LIN {X 14.324,Y -289.646,Z 149.698,A 92.831,B 90.000,C 0.000} C_DIS
LIN {X 14.364,Y -289.644,Z 149.777,A 92.839,B 90.000,C 0.000} C_DIS
LIN {X 14.595,Y -289.632,Z 150.119,A 92.885,B 90.000,C 0.000} C_DIS
LIN {X 14.694,Y -289.627,Z 150.212,A 92.904,B 90.000,C 0.000} C_DIS
LIN {X 14.908,Y -289.617,Z 150.520,A 92.947,B 90.000,C 0.000} C_DIS
LIN {X 16.420,Y -289.535,Z 152.509,A 93.246,B 90.000,C 0.000} C_DIS
LIN {X 16.512,Y -289.530,Z 152.653,A 93.264,B 90.000,C 0.000} C_DIS
LIN {X 18.087,Y -289.435,Z 154.593,A 93.576,B 90.000,C 0.000} C_DIS
LIN {X 18.457,Y -289.412,Z 155.070,A 93.649,B 90.000,C 0.000} C_DIS
LIN {X 18.491,Y -289.410,Z 155.103,A 93.656,B 90.000,C 0.000} C_DIS
LIN {X 18.557,Y -289.406,Z 155.188,A 93.669,B 90.000,C 0.000} C_DIS
LIN {X 18.610,Y -289.402,Z 155.273,A 93.679,B 90.000,C 0.000} C_DIS
LIN {X 18.698,Y -289.397,Z 155.384,A 93.697,B 90.000,C 0.000} C_DIS
LIN {X 18.848,Y -289.387,Z 155.532,A 93.726,B 90.000,C 0.000} C_DIS
LIN {X 18.933,Y -289.381,Z 155.598,A 93.743,B 90.000,C 0.000} C_DIS
LIN {X 18.971,Y -289.379,Z 155.701,A 93.751,B 90.000,C 0.000} C_DIS
LIN {X 20.031,Y -289.307,Z 156.976,A 93.961,B 90.000,C 0.000} C_DIS
LIN {X 20.180,Y -289.297,Z 157.094,A 93.990,B 90.000,C 0.000} C_DIS
LIN {X 20.232,Y -289.293,Z 157.151,A 94.000,B 90.000,C 0.000} C_DIS
LIN {X 20.247,Y -289.292,Z 157.208,A 94.004,B 90.000,C 0.000} C_DIS
LIN {X 20.626,Y -289.266,Z 157.610,A 94.079,B 90.000,C 0.000} C_DIS
LIN {X 20.742,Y -289.257,Z 157.720,A 94.102,B 90.000,C 0.000} C_DIS
LIN {X 20.768,Y -289.255,Z 157.777,A 94.107,B 90.000,C 0.000} C_DIS
LIN {X 21.906,Y -289.171,Z 158.799,A 94.332,B 90.000,C 0.000} C_DIS
LIN {X 22.359,Y -289.137,Z 159.201,A 94.422,B 90.000,C 0.000} C_DIS
LIN {X 23.494,Y -289.047,Z 160.165,A 94.647,B 90.000,C 0.000} C_DIS
LIN {X 23.807,Y -289.021,Z 160.394,A 94.709,B 90.000,C 0.000} C_DIS
LIN {X 23.862,Y -289.017,Z 160.451,A 94.720,B 90.000,C 0.000} C_DIS
LIN {X 23.876,Y -289.015,Z 160.508,A 94.723,B 90.000,C 0.000} C_DIS
LIN {X 24.686,Y -288.947,Z 161.134,A 94.883,B 90.000,C 0.000} C_DIS
LIN {X 24.833,Y -288.935,Z 161.286,A 94.912,B 90.000,C 0.000} C_DIS
LIN {X 25.476,Y -288.879,Z 161.759,A 95.040,B 90.000,C 0.000} C_DIS
LIN {X 25.535,Y -288.874,Z 161.845,A 95.051,B 90.000,C 0.000} C_DIS
LIN {X 25.733,Y -288.856,Z 161.987,A 95.091,B 90.000,C 0.000} C_DIS
LIN {X 25.749,Y -288.855,Z 162.044,A 95.094,B 90.000,C 0.000} C_DIS
LIN {X 26.204,Y -288.814,Z 162.384,A 95.184,B 90.000,C 0.000} C_DIS
LIN {X 26.243,Y -288.810,Z 162.442,A 95.192,B 90.000,C 0.000} C_DIS
LIN {X 26.264,Y -288.808,Z 162.499,A 95.196,B 90.000,C 0.000} C_DIS
LIN {X 27.201,Y -288.721,Z 163.333,A 95.382,B 90.000,C 0.000} C_DIS
LIN {X 29.132,Y -288.533,Z 164.205,A 95.765,B 90.000,C 0.000} C_DIS
LIN {X 31.516,Y -288.282,Z 164.913,A 96.239,B 90.000,C 0.000} C_DIS
LIN {X 33.522,Y -288.056,Z 165.228,A 96.638,B 90.000,C 0.000} C_DIS
LIN {X 36.003,Y -287.754,Z 165.278,A 97.132,B 90.000,C 0.000} C_DIS
LIN {X 37.185,Y -287.606,Z 165.298,A 97.367,B 90.000,C 0.000} C_DIS
LIN {X 38.173,Y -287.477,Z 165.175,A 97.564,B 90.000,C 0.000} C_DIS
LIN {X 39.512,Y -287.296,Z 164.884,A 97.831,B 90.000,C 0.000} C_DIS
LIN {X 39.611,Y -287.282,Z 164.845,A 97.850,B 90.000,C 0.000} C_DIS
LIN {X 40.343,Y -287.180,Z 164.702,A 97.997,B 90.000,C 0.000} C_DIS
LIN {X 40.569,Y -287.148,Z 164.621,A 98.042,B 90.000,C 0.000} C_DIS
LIN {X 40.681,Y -287.132,Z 164.611,A 98.064,B 90.000,C 0.000} C_DIS
LIN {X 42.877,Y -286.813,Z 163.977,A 98.502,B 90.000,C 0.000} C_DIS
LIN {X 42.990,Y -286.796,Z 163.962,A 98.525,B 90.000,C 0.000} C_DIS
LIN {X 43.102,Y -286.779,Z 163.932,A 98.547,B 90.000,C 0.000} C_DIS
LIN {X 43.758,Y -286.680,Z 163.656,A 98.678,B 90.000,C 0.000} C_DIS
LIN {X 43.856,Y -286.665,Z 163.644,A 98.698,B 90.000,C 0.000} C_DIS
LIN {X 46.143,Y -286.306,Z 162.699,A 99.155,B 90.000,C 0.000} C_DIS
LIN {X 46.563,Y -286.237,Z 162.499,A 99.240,B 90.000,C 0.000} C_DIS
LIN {X 47.119,Y -286.147,Z 162.115,A 99.351,B 90.000,C 0.000} C_DIS
LIN {X 47.257,Y -286.124,Z 162.044,A 99.378,B 90.000,C 0.000} C_DIS
LIN {X 47.317,Y -286.114,Z 161.984,A 99.391,B 90.000,C 0.000} C_DIS
LIN {X 48.334,Y -285.944,Z 161.191,A 99.594,B 90.000,C 0.000} C_DIS
LIN {X 48.383,Y -285.935,Z 161.105,A 99.604,B 90.000,C 0.000} C_DIS
LIN {X 48.468,Y -285.921,Z 161.020,A 99.621,B 90.000,C 0.000} C_DIS
LIN {X 48.552,Y -285.907,Z 160.953,A 99.638,B 90.000,C 0.000} C_DIS
LIN {X 48.585,Y -285.901,Z 160.921,A 99.644,B 90.000,C 0.000} C_DIS
LIN {X 50.411,Y -285.585,Z 159.243,A 100.011,B 90.000,C 0.000} C_DIS
LIN {X 50.514,Y -285.567,Z 159.135,A 100.031,B 90.000,C 0.000} C_DIS
LIN {X 50.570,Y -285.557,Z 159.114,A 100.043,B 90.000,C 0.000} C_DIS
LIN {X 50.626,Y -285.547,Z 159.064,A 100.054,B 90.000,C 0.000} C_DIS
LIN {X 51.727,Y -285.349,Z 156.829,A 100.275,B 90.000,C 0.000} C_DIS
LIN {X 51.777,Y -285.340,Z 156.731,A 100.285,B 90.000,C 0.000} C_DIS
LIN {X 52.198,Y -285.264,Z 155.800,A 100.369,B 90.000,C 0.000} C_DIS
LIN {X 52.229,Y -285.258,Z 155.405,A 100.376,B 90.000,C 0.000} C_DIS
LIN {X 52.149,Y -285.273,Z 155.422,A 100.359,B 90.000,C 0.000} C_DIS
LIN {X 51.928,Y -285.313,Z 155.589,A 100.315,B 90.000,C 0.000} C_DIS
LIN {X 51.746,Y -285.346,Z 155.763,A 100.279,B 90.000,C 0.000} C_DIS
LIN {X 51.520,Y -285.387,Z 156.070,A 100.233,B 90.000,C 0.000} C_DIS
LIN {X 51.426,Y -285.404,Z 156.169,A 100.214,B 90.000,C 0.000} C_DIS
LIN {X 51.130,Y -285.457,Z 156.551,A 100.155,B 90.000,C 0.000} C_DIS
LIN {X 50.883,Y -285.501,Z 156.767,A 100.105,B 90.000,C 0.000} C_DIS
LIN {X 50.632,Y -285.546,Z 157.151,A 100.055,B 90.000,C 0.000} C_DIS
LIN {X 48.944,Y -285.840,Z 158.739,A 99.717,B 90.000,C 0.000} C_DIS
LIN {X 48.327,Y -285.945,Z 159.090,A 99.593,B 90.000,C 0.000} C_DIS
LIN {X 48.215,Y -285.964,Z 159.139,A 99.570,B 90.000,C 0.000} C_DIS
LIN {X 48.131,Y -285.978,Z 159.199,A 99.554,B 90.000,C 0.000} C_DIS
LIN {X 48.047,Y -285.992,Z 159.243,A 99.537,B 90.000,C 0.000} C_DIS
LIN {X 47.103,Y -286.149,Z 159.921,A 99.348,B 90.000,C 0.000} C_DIS
LIN {X 46.868,Y -286.188,Z 160.040,A 99.301,B 90.000,C 0.000} C_DIS
LIN {X 46.475,Y -286.252,Z 160.349,A 99.222,B 90.000,C 0.000} C_DIS
LIN {X 46.419,Y -286.261,Z 160.366,A 99.211,B 90.000,C 0.000} C_DIS
LIN {X 46.363,Y -286.270,Z 160.391,A 99.199,B 90.000,C 0.000} C_DIS
LIN {X 46.283,Y -286.283,Z 160.451,A 99.183,B 90.000,C 0.000} C_DIS
LIN {X 45.576,Y -286.396,Z 160.853,A 99.042,B 90.000,C 0.000} C_DIS
LIN {X 44.677,Y -286.538,Z 161.257,A 98.862,B 90.000,C 0.000} C_DIS
LIN {X 44.565,Y -286.555,Z 161.295,A 98.840,B 90.000,C 0.000} C_DIS
LIN {X 43.565,Y -286.709,Z 161.759,A 98.640,B 90.000,C 0.000} C_DIS
LIN {X 41.526,Y -287.011,Z 162.566,A 98.233,B 90.000,C 0.000} C_DIS
LIN {X 41.301,Y -287.044,Z 162.601,A 98.188,B 90.000,C 0.000} C_DIS
LIN {X 40.977,Y -287.090,Z 162.722,A 98.123,B 90.000,C 0.000} C_DIS
LIN {X 38.530,Y -287.429,Z 163.103,A 97.635,B 90.000,C 0.000} C_DIS
LIN {X 37.750,Y -287.533,Z 163.175,A 97.480,B 90.000,C 0.000} C_DIS
LIN {X 35.270,Y -287.846,Z 163.117,A 96.986,B 90.000,C 0.000} C_DIS
LIN {X 32.811,Y -288.137,Z 162.780,A 96.496,B 90.000,C 0.000} C_DIS
LIN {X 30.430,Y -288.399,Z 162.061,A 96.023,B 90.000,C 0.000} C_DIS
LIN {X 29.103,Y -288.536,Z 161.533,A 95.760,B 90.000,C 0.000} C_DIS
LIN {X 28.948,Y -288.552,Z 161.424,A 95.729,B 90.000,C 0.000} C_DIS
LIN {X 28.296,Y -288.616,Z 161.071,A 95.599,B 90.000,C 0.000} C_DIS
LIN {X 28.141,Y -288.631,Z 160.962,A 95.569,B 90.000,C 0.000} C_DIS
LIN {X 27.574,Y -288.686,Z 160.678,A 95.456,B 90.000,C 0.000} C_DIS
LIN {X 27.006,Y -288.740,Z 160.337,A 95.343,B 90.000,C 0.000} C_DIS
LIN {X 26.825,Y -288.757,Z 160.259,A 95.307,B 90.000,C 0.000} C_DIS
LIN {X 26.623,Y -288.775,Z 160.142,A 95.267,B 90.000,C 0.000} C_DIS
LIN {X 26.439,Y -288.792,Z 159.996,A 95.231,B 90.000,C 0.000} C_DIS
LIN {X 25.672,Y -288.861,Z 159.484,A 95.079,B 90.000,C 0.000} C_DIS
LIN {X 25.308,Y -288.894,Z 159.140,A 95.007,B 90.000,C 0.000} C_DIS
LIN {X 24.741,Y -288.943,Z 158.391,A 94.894,B 90.000,C 0.000} C_DIS
LIN {X 24.666,Y -288.949,Z 158.346,A 94.879,B 90.000,C 0.000} C_DIS
LIN {X 23.494,Y -289.047,Z 157.203,A 94.647,B 90.000,C 0.000} C_DIS
LIN {X 22.038,Y -289.161,Z 155.956,A 94.358,B 90.000,C 0.000} C_DIS
LIN {X 21.452,Y -289.206,Z 155.331,A 94.242,B 90.000,C 0.000} C_DIS
LIN {X 21.337,Y -289.214,Z 155.245,A 94.219,B 90.000,C 0.000} C_DIS
LIN {X 21.256,Y -289.220,Z 155.155,A 94.203,B 90.000,C 0.000} C_DIS
LIN {X 21.228,Y -289.222,Z 155.103,A 94.198,B 90.000,C 0.000} C_DIS
LIN {X 21.168,Y -289.226,Z 155.043,A 94.186,B 90.000,C 0.000} C_DIS
LIN {X 20.955,Y -289.242,Z 154.735,A 94.144,B 90.000,C 0.000} C_DIS
LIN {X 20.884,Y -289.247,Z 154.595,A 94.130,B 90.000,C 0.000} C_DIS
LIN {X 20.824,Y -289.251,Z 154.534,A 94.118,B 90.000,C 0.000} C_DIS
LIN {X 20.799,Y -289.253,Z 154.477,A 94.113,B 90.000,C 0.000} C_DIS
LIN {X 20.786,Y -289.254,Z 154.420,A 94.110,B 90.000,C 0.000} C_DIS
LIN {X 20.630,Y -289.265,Z 154.235,A 94.079,B 90.000,C 0.000} C_DIS
LIN {X 19.990,Y -289.310,Z 153.410,A 93.953,B 90.000,C 0.000} C_DIS
LIN {X 19.863,Y -289.319,Z 153.211,A 93.927,B 90.000,C 0.000} C_DIS
LIN {X 18.387,Y -289.417,Z 151.407,A 93.635,B 90.000,C 0.000} C_DIS
LIN {X 18.287,Y -289.423,Z 151.314,A 93.615,B 90.000,C 0.000} C_DIS
LIN {X 16.924,Y -289.506,Z 149.655,A 93.346,B 90.000,C 0.000} C_DIS
LIN {X 16.797,Y -289.513,Z 149.456,A 93.320,B 90.000,C 0.000} C_DIS
LIN {X 16.711,Y -289.518,Z 149.413,A 93.304,B 90.000,C 0.000} C_DIS
LIN {X 16.626,Y -289.523,Z 149.330,A 93.287,B 90.000,C 0.000} C_DIS
LIN {X 15.149,Y -289.604,Z 147.315,A 92.994,B 90.000,C 0.000} C_DIS
LIN {X 14.736,Y -289.625,Z 146.796,A 92.913,B 90.000,C 0.000} C_DIS
LIN {X 14.707,Y -289.627,Z 146.682,A 92.907,B 90.000,C 0.000} C_DIS
LIN {X 14.145,Y -289.655,Z 146.113,A 92.796,B 90.000,C 0.000} C_DIS
LIN {X 14.069,Y -289.659,Z 146.056,A 92.781,B 90.000,C 0.000} C_DIS
LIN {X 13.615,Y -289.680,Z 145.498,A 92.691,B 90.000,C 0.000} C_DIS
LIN {X 13.402,Y -289.690,Z 145.203,A 92.649,B 90.000,C 0.000} C_DIS
LIN {X 13.265,Y -289.696,Z 144.790,A 92.622,B 90.000,C 0.000} C_DIS
LIN {X 12.920,Y -289.712,Z 144.349,A 92.554,B 90.000,C 0.000} C_DIS
LIN {X 12.904,Y -289.713,Z 144.292,A 92.550,B 90.000,C 0.000} C_DIS
LIN {X 12.879,Y -289.714,Z 144.236,A 92.545,B 90.000,C 0.000} C_DIS
LIN {X 12.759,Y -289.719,Z 144.065,A 92.522,B 90.000,C 0.000} C_DIS
LIN {X 12.709,Y -289.721,Z 143.951,A 92.512,B 90.000,C 0.000} C_DIS
LIN {X 12.595,Y -289.726,Z 143.780,A 92.489,B 90.000,C 0.000} C_DIS
LIN {X 12.493,Y -289.731,Z 143.549,A 92.469,B 90.000,C 0.000} C_DIS
LIN {X 12.080,Y -289.748,Z 142.870,A 92.387,B 90.000,C 0.000} C_DIS
LIN {X 11.620,Y -289.767,Z 141.618,A 92.296,B 90.000,C 0.000} C_DIS
LIN {X 11.609,Y -289.768,Z 141.505,A 92.294,B 90.000,C 0.000} C_DIS
LIN {X 11.528,Y -289.771,Z 141.277,A 92.278,B 90.000,C 0.000} C_DIS
LIN {X 11.515,Y -289.771,Z 141.163,A 92.276,B 90.000,C 0.000} C_DIS
LIN {X 11.268,Y -289.781,Z 140.537,A 92.227,B 90.000,C 0.000} C_DIS
LIN {X 11.244,Y -289.782,Z 140.424,A 92.222,B 90.000,C 0.000} C_DIS
LIN {X 11.230,Y -289.782,Z 140.283,A 92.219,B 90.000,C 0.000} C_DIS
LIN {X 10.936,Y -289.794,Z 139.286,A 92.161,B 90.000,C 0.000} C_DIS
LIN {X 10.927,Y -289.794,Z 139.172,A 92.159,B 90.000,C 0.000} C_DIS
LIN {X 10.846,Y -289.797,Z 138.944,A 92.143,B 90.000,C 0.000} C_DIS
LIN {X 10.836,Y -289.798,Z 138.830,A 92.141,B 90.000,C 0.000} C_DIS
LIN {X 10.539,Y -289.808,Z 137.806,A 92.083,B 90.000,C 0.000} C_DIS
LIN {X 10.529,Y -289.809,Z 137.692,A 92.081,B 90.000,C 0.000} C_DIS
LIN {X 10.448,Y -289.812,Z 137.465,A 92.065,B 90.000,C 0.000} C_DIS
LIN {X 10.438,Y -289.812,Z 137.351,A 92.063,B 90.000,C 0.000} C_DIS
LIN {X 10.086,Y -289.825,Z 136.099,A 91.993,B 90.000,C 0.000} C_DIS
LIN {X 10.074,Y -289.825,Z 135.986,A 91.991,B 90.000,C 0.000} C_DIS
LIN {X 9.993,Y -289.828,Z 135.758,A 91.975,B 90.000,C 0.000} C_DIS
LIN {X 9.979,Y -289.828,Z 135.617,A 91.972,B 90.000,C 0.000} C_DIS
LIN {X 9.688,Y -289.838,Z 134.620,A 91.915,B 90.000,C 0.000} C_DIS
LIN {X 9.676,Y -289.839,Z 134.506,A 91.912,B 90.000,C 0.000} C_DIS
LIN {X 9.595,Y -289.841,Z 134.279,A 91.896,B 90.000,C 0.000} C_DIS
LIN {X 9.583,Y -289.842,Z 134.165,A 91.894,B 90.000,C 0.000} C_DIS
LIN {X 9.298,Y -289.851,Z 133.255,A 91.837,B 90.000,C 0.000} C_DIS
LIN {X 9.059,Y -289.858,Z 132.515,A 91.790,B 90.000,C 0.000} C_DIS
LIN {X 9.010,Y -289.860,Z 132.287,A 91.780,B 90.000,C 0.000} C_DIS
LIN {X 8.778,Y -289.867,Z 131.662,A 91.735,B 90.000,C 0.000} C_DIS
LIN {X 8.743,Y -289.868,Z 131.434,A 91.728,B 90.000,C 0.000} C_DIS
LIN {X 8.427,Y -289.878,Z 130.524,A 91.665,B 90.000,C 0.000} C_DIS
LIN {X 8.385,Y -289.879,Z 130.296,A 91.657,B 90.000,C 0.000} C_DIS
LIN {X 8.155,Y -289.885,Z 129.556,A 91.612,B 90.000,C 0.000} C_DIS
LIN {X 8.140,Y -289.886,Z 129.443,A 91.608,B 90.000,C 0.000} C_DIS
LIN {X 8.066,Y -289.888,Z 129.236,A 91.594,B 90.000,C 0.000} C_DIS
LIN {X 7.584,Y -289.901,Z 127.235,A 91.499,B 90.000,C 0.000} C_DIS
LIN {X 7.572,Y -289.901,Z 127.107,A 91.496,B 90.000,C 0.000} C_DIS
LIN {X 7.491,Y -289.903,Z 126.882,A 91.480,B 90.000,C 0.000} C_DIS
LIN {X 7.481,Y -289.903,Z 126.768,A 91.478,B 90.000,C 0.000} C_DIS
LIN {X 7.127,Y -289.912,Z 125.517,A 91.408,B 90.000,C 0.000} C_DIS
LIN {X 6.731,Y -289.922,Z 124.037,A 91.330,B 90.000,C 0.000} C_DIS
LIN {X 6.351,Y -289.930,Z 122.795,A 91.255,B 90.000,C 0.000} C_DIS
LIN {X 6.337,Y -289.931,Z 122.672,A 91.252,B 90.000,C 0.000} C_DIS
LIN {X 6.102,Y -289.936,Z 121.932,A 91.206,B 90.000,C 0.000} C_DIS
LIN {X 6.053,Y -289.937,Z 121.705,A 91.196,B 90.000,C 0.000} C_DIS
LIN {X 5.809,Y -289.942,Z 121.079,A 91.148,B 90.000,C 0.000} C_DIS
LIN {X 5.766,Y -289.943,Z 120.851,A 91.139,B 90.000,C 0.000} C_DIS
LIN {X 5.306,Y -289.951,Z 119.566,A 91.048,B 90.000,C 0.000} C_DIS
LIN {X 5.289,Y -289.952,Z 119.471,A 91.045,B 90.000,C 0.000} C_DIS
LIN {X 4.887,Y -289.959,Z 118.362,A 90.966,B 90.000,C 0.000} C_DIS
LIN {X 4.789,Y -289.960,Z 118.177,A 90.946,B 90.000,C 0.000} C_DIS
LIN {X 4.760,Y -289.961,Z 118.063,A 90.941,B 90.000,C 0.000} C_DIS
LIN {X 4.745,Y -289.961,Z 117.950,A 90.937,B 90.000,C 0.000} C_DIS
LIN {X 3.807,Y -289.975,Z 115.632,A 90.752,B 90.000,C 0.000} C_DIS
LIN {X 2.964,Y -289.985,Z 113.398,A 90.586,B 90.000,C 0.000} C_DIS
LIN {X 2.920,Y -289.985,Z 113.170,A 90.577,B 90.000,C 0.000} C_DIS
LIN {X 2.749,Y -289.987,Z 112.772,A 90.543,B 90.000,C 0.000} C_DIS
LIN {X 2.695,Y -289.987,Z 112.544,A 90.532,B 90.000,C 0.000} C_DIS
LIN {X 2.522,Y -289.989,Z 112.146,A 90.498,B 90.000,C 0.000} C_DIS
LIN {X 2.467,Y -289.990,Z 111.919,A 90.487,B 90.000,C 0.000} C_DIS
LIN {X 2.288,Y -289.991,Z 111.520,A 90.452,B 90.000,C 0.000} C_DIS
LIN {X 2.253,Y -289.991,Z 111.407,A 90.445,B 90.000,C 0.000} C_DIS
LIN {X 1.843,Y -289.994,Z 110.382,A 90.364,B 90.000,C 0.000} C_DIS
LIN {X 1.785,Y -289.995,Z 110.155,A 90.353,B 90.000,C 0.000} C_DIS
LIN {X 1.605,Y -289.996,Z 109.757,A 90.317,B 90.000,C 0.000} C_DIS
LIN {X 1.567,Y -289.996,Z 109.643,A 90.310,B 90.000,C 0.000} C_DIS
LIN {X 1.388,Y -289.997,Z 109.245,A 90.274,B 90.000,C 0.000} C_DIS
LIN {X 1.333,Y -289.997,Z 109.017,A 90.263,B 90.000,C 0.000} C_DIS
LIN {X 1.162,Y -289.998,Z 108.619,A 90.230,B 90.000,C 0.000} C_DIS
LIN {X 1.116,Y -289.998,Z 108.391,A 90.220,B 90.000,C 0.000} C_DIS
LIN {X 0.935,Y -289.998,Z 107.993,A 90.185,B 90.000,C 0.000} C_DIS
LIN {X 0.915,Y -289.999,Z 107.879,A 90.181,B 90.000,C 0.000} C_DIS
LIN {X 0.835,Y -289.999,Z 107.651,A 90.165,B 90.000,C 0.000} C_DIS
LIN {X 0.822,Y -289.999,Z 107.538,A 90.162,B 90.000,C 0.000} C_DIS
LIN {X 0.578,Y -289.999,Z 106.876,A 90.114,B 90.000,C 0.000} C_DIS
LIN {X 0.545,Y -289.999,Z 106.627,A 90.108,B 90.000,C 0.000} C_DIS
LIN {X 0.301,Y -290.000,Z 105.913,A 90.060,B 90.000,C 0.000} C_DIS
LIN {X 0.252,Y -290.000,Z 105.660,A 90.050,B 90.000,C 0.000} C_DIS
LIN {X -0.043,Y -290.000,Z 104.773,A 89.992,B 90.000,C 0.000} C_DIS
LIN {X -0.385,Y -290.000,Z 103.555,A 89.924,B 90.000,C 0.000} C_DIS
LIN {X -0.393,Y -290.000,Z 103.441,A 89.922,B 90.000,C 0.000} C_DIS
LIN {X -0.474,Y -290.000,Z 103.214,A 89.906,B 90.000,C 0.000} C_DIS
LIN {X -0.489,Y -290.000,Z 103.100,A 89.903,B 90.000,C 0.000} C_DIS
LIN {X -0.560,Y -289.999,Z 102.943,A 89.889,B 90.000,C 0.000} C_DIS
LIN {X -0.949,Y -289.998,Z 101.234,A 89.812,B 90.000,C 0.000} C_DIS
LIN {X -0.961,Y -289.998,Z 101.106,A 89.810,B 90.000,C 0.000} C_DIS
LIN {X -1.033,Y -289.998,Z 100.886,A 89.796,B 90.000,C 0.000} C_DIS
LIN {X -1.049,Y -289.998,Z 100.745,A 89.793,B 90.000,C 0.000} C_DIS
LIN {X -1.351,Y -289.997,Z 99.743,A 89.733,B 90.000,C 0.000} C_DIS
LIN {X -1.360,Y -289.997,Z 99.629,A 89.731,B 90.000,C 0.000} C_DIS
LIN {X -1.441,Y -289.996,Z 99.402,A 89.715,B 90.000,C 0.000} C_DIS
LIN {X -1.452,Y -289.996,Z 99.288,A 89.713,B 90.000,C 0.000} C_DIS
LIN {X -1.701,Y -289.995,Z 98.618,A 89.664,B 90.000,C 0.000} C_DIS
LIN {X -1.735,Y -289.995,Z 98.411,A 89.657,B 90.000,C 0.000} C_DIS
LIN {X -2.039,Y -289.993,Z 97.524,A 89.597,B 90.000,C 0.000} C_DIS
LIN {X -2.067,Y -289.993,Z 97.410,A 89.592,B 90.000,C 0.000} C_DIS
LIN {X -2.078,Y -289.993,Z 97.296,A 89.589,B 90.000,C 0.000} C_DIS
LIN {X -2.316,Y -289.991,Z 96.557,A 89.543,B 90.000,C 0.000} C_DIS
LIN {X -2.410,Y -289.990,Z 96.053,A 89.524,B 90.000,C 0.000} C_DIS
LIN {X -2.876,Y -289.986,Z 94.338,A 89.432,B 90.000,C 0.000} C_DIS
LIN {X -3.082,Y -289.984,Z 93.840,A 89.391,B 90.000,C 0.000} C_DIS
LIN {X -3.621,Y -289.977,Z 91.399,A 89.285,B 90.000,C 0.000} C_DIS
LIN {X -3.625,Y -289.977,Z 91.365,A 89.284,B 90.000,C 0.000} C_DIS
LIN {X -3.668,Y -289.977,Z 91.265,A 89.275,B 90.000,C 0.000} C_DIS
LIN {X -3.693,Y -289.976,Z 91.152,A 89.270,B 90.000,C 0.000} C_DIS
LIN {X -3.731,Y -289.976,Z 91.038,A 89.263,B 90.000,C 0.000} C_DIS
LIN {X -3.782,Y -289.975,Z 90.696,A 89.253,B 90.000,C 0.000} C_DIS
LIN {X -3.934,Y -289.973,Z 90.264,A 89.223,B 90.000,C 0.000} C_DIS
LIN {X -4.021,Y -289.972,Z 89.548,A 89.205,B 90.000,C 0.000} C_DIS
LIN {X -3.846,Y -289.974,Z 87.324,A 89.240,B 90.000,C 0.000} C_DIS
LIN {X -3.625,Y -289.977,Z 86.490,A 89.284,B 90.000,C 0.000} C_DIS
LIN {X -2.878,Y -289.986,Z 84.495,A 89.431,B 90.000,C 0.000} C_DIS
LIN {X -2.858,Y -287.986,Z 84.495,A 89.431,B 90.000,C 0.000} C_DIS
WAIT SEC 0.1
RET=EKI_SetBool("oxy","torchState",FALSE)
RET = EKI_Send("oxy","torchState")
LIN {X -2.679,Y -269.987,Z 84.495,A 89.431,B 90.000,C 0.000} C_DIS
LIN {X 19.872,Y -269.268,Z 90.056,A 94.221,B 90.000,C 0.000} C_DIS
LIN {X 21.197,Y -287.219,Z 90.056,A 94.221,B 90.000,C 0.000} C_DIS
LIN {X 21.344,Y -289.213,Z 90.056,A 94.221,B 90.000,C 0.000} C_DIS
WAIT SEC 1
RET=EKI_SetBool("oxy","torchState",TRUE)
RET = EKI_Send("oxy","torchState")
LIN {X 21.267,Y -289.219,Z 90.801,A 94.206,B 90.000,C 0.000} C_DIS
LIN {X 21.412,Y -289.208,Z 91.457,A 94.234,B 90.000,C 0.000} C_DIS
LIN {X 21.508,Y -289.201,Z 91.574,A 94.253,B 90.000,C 0.000} C_DIS
LIN {X 21.583,Y -289.196,Z 91.731,A 94.268,B 90.000,C 0.000} C_DIS
LIN {X 21.758,Y -289.183,Z 91.977,A 94.303,B 90.000,C 0.000} C_DIS
LIN {X 22.084,Y -289.158,Z 92.312,A 94.367,B 90.000,C 0.000} C_DIS
LIN {X 22.414,Y -289.133,Z 92.517,A 94.433,B 90.000,C 0.000} C_DIS
LIN {X 22.473,Y -289.128,Z 92.572,A 94.444,B 90.000,C 0.000} C_DIS
LIN {X 23.360,Y -289.058,Z 92.826,A 94.620,B 90.000,C 0.000} C_DIS
LIN {X 23.777,Y -289.024,Z 92.846,A 94.703,B 90.000,C 0.000} C_DIS
LIN {X 24.514,Y -288.962,Z 92.716,A 94.849,B 90.000,C 0.000} C_DIS
LIN {X 24.628,Y -288.952,Z 92.694,A 94.872,B 90.000,C 0.000} C_DIS
LIN {X 25.648,Y -288.864,Z 92.287,A 95.074,B 90.000,C 0.000} C_DIS
LIN {X 25.691,Y -288.860,Z 92.242,A 95.082,B 90.000,C 0.000} C_DIS
LIN {X 26.130,Y -288.820,Z 92.119,A 95.170,B 90.000,C 0.000} C_DIS
LIN {X 26.244,Y -288.810,Z 92.061,A 95.192,B 90.000,C 0.000} C_DIS
LIN {X 26.332,Y -288.802,Z 92.036,A 95.210,B 90.000,C 0.000} C_DIS
LIN {X 26.781,Y -288.761,Z 91.837,A 95.299,B 90.000,C 0.000} C_DIS
LIN {X 27.008,Y -288.740,Z 91.793,A 95.344,B 90.000,C 0.000} C_DIS
LIN {X 28.877,Y -288.559,Z 91.089,A 95.715,B 90.000,C 0.000} C_DIS
LIN {X 29.103,Y -288.536,Z 91.037,A 95.760,B 90.000,C 0.000} C_DIS
LIN {X 29.499,Y -288.496,Z 90.863,A 95.838,B 90.000,C 0.000} C_DIS
LIN {X 29.669,Y -288.478,Z 90.825,A 95.872,B 90.000,C 0.000} C_DIS
LIN {X 30.914,Y -288.348,Z 90.347,A 96.119,B 90.000,C 0.000} C_DIS
LIN {X 31.140,Y -288.323,Z 90.308,A 96.164,B 90.000,C 0.000} C_DIS
LIN {X 31.536,Y -288.280,Z 90.130,A 96.243,B 90.000,C 0.000} C_DIS
LIN {X 31.763,Y -288.255,Z 90.086,A 96.288,B 90.000,C 0.000} C_DIS
LIN {X 33.542,Y -288.054,Z 89.445,A 96.642,B 90.000,C 0.000} C_DIS
LIN {X 33.628,Y -288.044,Z 89.393,A 96.659,B 90.000,C 0.000} C_DIS
LIN {X 33.854,Y -288.017,Z 89.343,A 96.704,B 90.000,C 0.000} C_DIS
LIN {X 34.677,Y -287.919,Z 88.990,A 96.868,B 90.000,C 0.000} C_DIS
LIN {X 34.791,Y -287.905,Z 88.890,A 96.890,B 90.000,C 0.000} C_DIS
LIN {X 35.130,Y -287.864,Z 88.663,A 96.958,B 90.000,C 0.000} C_DIS
LIN {X 35.547,Y -287.813,Z 88.136,A 97.041,B 90.000,C 0.000} C_DIS
LIN {X 35.761,Y -287.787,Z 87.490,A 97.083,B 90.000,C 0.000} C_DIS
LIN {X 35.859,Y -287.774,Z 86.829,A 97.103,B 90.000,C 0.000} C_DIS
LIN {X 35.778,Y -287.785,Z 86.315,A 97.087,B 90.000,C 0.000} C_DIS
LIN {X 35.744,Y -287.789,Z 86.262,A 97.080,B 90.000,C 0.000} C_DIS
LIN {X 35.719,Y -287.792,Z 86.174,A 97.075,B 90.000,C 0.000} C_DIS
LIN {X 35.549,Y -287.813,Z 85.803,A 97.041,B 90.000,C 0.000} C_DIS
LIN {X 35.436,Y -287.827,Z 85.622,A 97.019,B 90.000,C 0.000} C_DIS
LIN {X 34.862,Y -287.897,Z 85.064,A 96.904,B 90.000,C 0.000} C_DIS
LIN {X 34.722,Y -287.914,Z 84.978,A 96.877,B 90.000,C 0.000} C_DIS
LIN {X 34.419,Y -287.950,Z 84.838,A 96.816,B 90.000,C 0.000} C_DIS
LIN {X 33.782,Y -288.026,Z 84.659,A 96.690,B 90.000,C 0.000} C_DIS
LIN {X 32.950,Y -288.122,Z 84.682,A 96.524,B 90.000,C 0.000} C_DIS
LIN {X 32.745,Y -288.145,Z 84.756,A 96.483,B 90.000,C 0.000} C_DIS
LIN {X 32.589,Y -288.163,Z 84.770,A 96.452,B 90.000,C 0.000} C_DIS
LIN {X 30.253,Y -288.418,Z 85.623,A 95.988,B 90.000,C 0.000} C_DIS
LIN {X 30.136,Y -288.430,Z 85.658,A 95.965,B 90.000,C 0.000} C_DIS
LIN {X 28.707,Y -288.576,Z 86.217,A 95.681,B 90.000,C 0.000} C_DIS
LIN {X 28.480,Y -288.598,Z 86.261,A 95.636,B 90.000,C 0.000} C_DIS
LIN {X 27.547,Y -288.689,Z 86.600,A 95.451,B 90.000,C 0.000} C_DIS
LIN {X 27.461,Y -288.697,Z 86.660,A 95.434,B 90.000,C 0.000} C_DIS
LIN {X 26.863,Y -288.753,Z 86.890,A 95.315,B 90.000,C 0.000} C_DIS
LIN {X 24.855,Y -288.933,Z 87.640,A 94.917,B 90.000,C 0.000} C_DIS
LIN {X 24.628,Y -288.952,Z 87.681,A 94.872,B 90.000,C 0.000} C_DIS
LIN {X 23.960,Y -289.008,Z 87.924,A 94.739,B 90.000,C 0.000} C_DIS
LIN {X 23.754,Y -289.025,Z 87.956,A 94.698,B 90.000,C 0.000} C_DIS
LIN {X 22.857,Y -289.098,Z 88.307,A 94.521,B 90.000,C 0.000} C_DIS
LIN {X 22.757,Y -289.106,Z 88.364,A 94.501,B 90.000,C 0.000} C_DIS
LIN {X 22.680,Y -289.112,Z 88.421,A 94.486,B 90.000,C 0.000} C_DIS
LIN {X 22.079,Y -289.158,Z 88.789,A 94.366,B 90.000,C 0.000} C_DIS
LIN {X 21.677,Y -289.189,Z 89.207,A 94.287,B 90.000,C 0.000} C_DIS
LIN {X 21.499,Y -289.202,Z 89.445,A 94.251,B 90.000,C 0.000} C_DIS
LIN {X 21.344,Y -289.213,Z 90.056,A 94.221,B 90.000,C 0.000} C_DIS
LIN {X 21.197,Y -287.219,Z 90.056,A 94.221,B 90.000,C 0.000} C_DIS
WAIT SEC 0.1
RET=EKI_SetBool("oxy","torchState",FALSE)
RET = EKI_Send("oxy","torchState")
LIN {X 19.872,Y -269.268,Z 90.056,A 94.221,B 90.000,C 0.000} C_DIS
LIN {X 27.934,Y -268.551,Z 97.065,A 95.938,B 90.000,C 0.000} C_DIS
LIN {X 29.796,Y -286.454,Z 97.065,A 95.938,B 90.000,C 0.000} C_DIS
LIN {X 30.003,Y -288.444,Z 97.065,A 95.938,B 90.000,C 0.000} C_DIS
WAIT SEC 1
RET=EKI_SetBool("oxy","torchState",TRUE)
RET = EKI_Send("oxy","torchState")
LIN {X 30.462,Y -288.396,Z 96.489,A 96.029,B 90.000,C 0.000} C_DIS
LIN {X 30.518,Y -288.390,Z 96.471,A 96.041,B 90.000,C 0.000} C_DIS
LIN {X 30.575,Y -288.384,Z 96.416,A 96.052,B 90.000,C 0.000} C_DIS
LIN {X 30.660,Y -288.375,Z 96.293,A 96.069,B 90.000,C 0.000} C_DIS
LIN {X 30.744,Y -288.366,Z 96.207,A 96.086,B 90.000,C 0.000} C_DIS
LIN {X 31.197,Y -288.317,Z 95.592,A 96.176,B 90.000,C 0.000} C_DIS
LIN {X 31.425,Y -288.292,Z 95.305,A 96.221,B 90.000,C 0.000} C_DIS
LIN {X 31.519,Y -288.282,Z 95.213,A 96.239,B 90.000,C 0.000} C_DIS
LIN {X 31.989,Y -288.230,Z 94.568,A 96.333,B 90.000,C 0.000} C_DIS
LIN {X 32.141,Y -288.213,Z 94.416,A 96.363,B 90.000,C 0.000} C_DIS
LIN {X 33.696,Y -288.036,Z 92.467,A 96.672,B 90.000,C 0.000} C_DIS
LIN {X 33.743,Y -288.030,Z 92.403,A 96.682,B 90.000,C 0.000} C_DIS
LIN {X 33.839,Y -288.019,Z 92.305,A 96.701,B 90.000,C 0.000} C_DIS
LIN {X 34.306,Y -287.964,Z 91.712,A 96.794,B 90.000,C 0.000} C_DIS
LIN {X 34.758,Y -287.909,Z 91.091,A 96.884,B 90.000,C 0.000} C_DIS
LIN {X 34.843,Y -287.899,Z 91.002,A 96.901,B 90.000,C 0.000} C_DIS
LIN {X 34.986,Y -287.882,Z 90.810,A 96.929,B 90.000,C 0.000} C_DIS
LIN {X 36.291,Y -287.720,Z 89.937,A 97.189,B 90.000,C 0.000} C_DIS
LIN {X 37.041,Y -287.625,Z 89.877,A 97.338,B 90.000,C 0.000} C_DIS
LIN {X 37.672,Y -287.543,Z 90.010,A 97.464,B 90.000,C 0.000} C_DIS
LIN {X 37.989,Y -287.501,Z 90.127,A 97.527,B 90.000,C 0.000} C_DIS
LIN {X 38.088,Y -287.488,Z 90.186,A 97.547,B 90.000,C 0.000} C_DIS
LIN {X 38.652,Y -287.413,Z 90.666,A 97.659,B 90.000,C 0.000} C_DIS
LIN {X 38.864,Y -287.384,Z 90.950,A 97.702,B 90.000,C 0.000} C_DIS
LIN {X 39.015,Y -287.364,Z 91.225,A 97.732,B 90.000,C 0.000} C_DIS
LIN {X 39.198,Y -287.339,Z 91.820,A 97.768,B 90.000,C 0.000} C_DIS
LIN {X 39.176,Y -287.342,Z 92.659,A 97.764,B 90.000,C 0.000} C_DIS
LIN {X 39.011,Y -287.364,Z 93.160,A 97.731,B 90.000,C 0.000} C_DIS
LIN {X 38.653,Y -287.412,Z 93.752,A 97.660,B 90.000,C 0.000} C_DIS
LIN {X 38.596,Y -287.420,Z 93.874,A 97.648,B 90.000,C 0.000} C_DIS
LIN {X 38.511,Y -287.432,Z 93.960,A 97.631,B 90.000,C 0.000} C_DIS
LIN {X 38.427,Y -287.443,Z 94.083,A 97.614,B 90.000,C 0.000} C_DIS
LIN {X 38.370,Y -287.450,Z 94.139,A 97.603,B 90.000,C 0.000} C_DIS
LIN {X 38.314,Y -287.458,Z 94.159,A 97.592,B 90.000,C 0.000} C_DIS
LIN {X 37.754,Y -287.532,Z 94.839,A 97.480,B 90.000,C 0.000} C_DIS
LIN {X 37.631,Y -287.548,Z 94.931,A 97.456,B 90.000,C 0.000} C_DIS
LIN {X 37.383,Y -287.580,Z 95.249,A 97.406,B 90.000,C 0.000} C_DIS
LIN {X 37.295,Y -287.592,Z 95.331,A 97.389,B 90.000,C 0.000} C_DIS
LIN {X 37.158,Y -287.610,Z 95.533,A 97.362,B 90.000,C 0.000} C_DIS
LIN {X 37.073,Y -287.621,Z 95.592,A 97.345,B 90.000,C 0.000} C_DIS
LIN {X 37.015,Y -287.628,Z 95.720,A 97.333,B 90.000,C 0.000} C_DIS
LIN {X 36.734,Y -287.664,Z 96.114,A 97.277,B 90.000,C 0.000} C_DIS
LIN {X 36.678,Y -287.671,Z 96.130,A 97.266,B 90.000,C 0.000} C_DIS
LIN {X 36.537,Y -287.689,Z 96.329,A 97.238,B 90.000,C 0.000} C_DIS
LIN {X 36.452,Y -287.700,Z 96.388,A 97.221,B 90.000,C 0.000} C_DIS
LIN {X 36.395,Y -287.707,Z 96.516,A 97.210,B 90.000,C 0.000} C_DIS
LIN {X 36.113,Y -287.743,Z 96.910,A 97.154,B 90.000,C 0.000} C_DIS
LIN {X 36.057,Y -287.750,Z 96.927,A 97.142,B 90.000,C 0.000} C_DIS
LIN {X 36.000,Y -287.757,Z 96.982,A 97.131,B 90.000,C 0.000} C_DIS
LIN {X 35.916,Y -287.767,Z 97.105,A 97.114,B 90.000,C 0.000} C_DIS
LIN {X 35.831,Y -287.778,Z 97.191,A 97.097,B 90.000,C 0.000} C_DIS
LIN {X 35.774,Y -287.785,Z 97.313,A 97.086,B 90.000,C 0.000} C_DIS
LIN {X 35.492,Y -287.820,Z 97.707,A 97.030,B 90.000,C 0.000} C_DIS
LIN {X 35.436,Y -287.827,Z 97.723,A 97.019,B 90.000,C 0.000} C_DIS
LIN {X 35.379,Y -287.834,Z 97.778,A 97.007,B 90.000,C 0.000} C_DIS
LIN {X 35.295,Y -287.844,Z 97.902,A 96.991,B 90.000,C 0.000} C_DIS
LIN {X 35.210,Y -287.855,Z 97.988,A 96.974,B 90.000,C 0.000} C_DIS
LIN {X 34.758,Y -287.909,Z 98.599,A 96.884,B 90.000,C 0.000} C_DIS
LIN {X 33.685,Y -288.037,Z 99.962,A 96.670,B 90.000,C 0.000} C_DIS
LIN {X 33.600,Y -288.047,Z 100.048,A 96.653,B 90.000,C 0.000} C_DIS
LIN {X 33.515,Y -288.057,Z 100.171,A 96.636,B 90.000,C 0.000} C_DIS
LIN {X 33.459,Y -288.063,Z 100.227,A 96.625,B 90.000,C 0.000} C_DIS
LIN {X 33.402,Y -288.070,Z 100.243,A 96.614,B 90.000,C 0.000} C_DIS
LIN {X 33.121,Y -288.102,Z 100.637,A 96.558,B 90.000,C 0.000} C_DIS
LIN {X 33.063,Y -288.109,Z 100.765,A 96.547,B 90.000,C 0.000} C_DIS
LIN {X 32.978,Y -288.119,Z 100.824,A 96.530,B 90.000,C 0.000} C_DIS
LIN {X 32.841,Y -288.134,Z 101.026,A 96.502,B 90.000,C 0.000} C_DIS
LIN {X 32.752,Y -288.145,Z 101.108,A 96.485,B 90.000,C 0.000} C_DIS
LIN {X 32.582,Y -288.164,Z 101.337,A 96.451,B 90.000,C 0.000} C_DIS
LIN {X 32.441,Y -288.180,Z 101.477,A 96.423,B 90.000,C 0.000} C_DIS
LIN {X 32.356,Y -288.189,Z 101.600,A 96.406,B 90.000,C 0.000} C_DIS
LIN {X 32.271,Y -288.199,Z 101.686,A 96.389,B 90.000,C 0.000} C_DIS
LIN {X 31.367,Y -288.299,Z 102.819,A 96.209,B 90.000,C 0.000} C_DIS
LIN {X 30.900,Y -288.349,Z 103.387,A 96.117,B 90.000,C 0.000} C_DIS
LIN {X 30.744,Y -288.366,Z 103.642,A 96.086,B 90.000,C 0.000} C_DIS
LIN {X 30.660,Y -288.375,Z 103.726,A 96.069,B 90.000,C 0.000} C_DIS
LIN {X 30.575,Y -288.384,Z 103.785,A 96.052,B 90.000,C 0.000} C_DIS
LIN {X 29.216,Y -288.525,Z 105.544,A 95.782,B 90.000,C 0.000} C_DIS
LIN {X 29.132,Y -288.533,Z 105.603,A 95.765,B 90.000,C 0.000} C_DIS
LIN {X 29.047,Y -288.542,Z 105.686,A 95.748,B 90.000,C 0.000} C_DIS
LIN {X 28.891,Y -288.557,Z 105.943,A 95.718,B 90.000,C 0.000} C_DIS
LIN {X 28.580,Y -288.588,Z 106.288,A 95.656,B 90.000,C 0.000} C_DIS
LIN {X 28.424,Y -288.604,Z 106.517,A 95.625,B 90.000,C 0.000} C_DIS
LIN {X 28.254,Y -288.620,Z 106.693,A 95.591,B 90.000,C 0.000} C_DIS
LIN {X 27.518,Y -288.691,Z 107.643,A 95.445,B 90.000,C 0.000} C_DIS
LIN {X 27.348,Y -288.708,Z 107.818,A 95.411,B 90.000,C 0.000} C_DIS
LIN {X 26.895,Y -288.750,Z 108.446,A 95.321,B 90.000,C 0.000} C_DIS
LIN {X 26.725,Y -288.766,Z 108.564,A 95.288,B 90.000,C 0.000} C_DIS
LIN {X 26.667,Y -288.771,Z 108.692,A 95.276,B 90.000,C 0.000} C_DIS
LIN {X 26.385,Y -288.797,Z 109.086,A 95.220,B 90.000,C 0.000} C_DIS
LIN {X 26.328,Y -288.802,Z 109.102,A 95.209,B 90.000,C 0.000} C_DIS
LIN {X 26.271,Y -288.808,Z 109.158,A 95.198,B 90.000,C 0.000} C_DIS
LIN {X 26.186,Y -288.815,Z 109.281,A 95.181,B 90.000,C 0.000} C_DIS
LIN {X 26.101,Y -288.823,Z 109.369,A 95.164,B 90.000,C 0.000} C_DIS
LIN {X 26.031,Y -288.829,Z 109.498,A 95.150,B 90.000,C 0.000} C_DIS
LIN {X 25.719,Y -288.857,Z 109.902,A 95.088,B 90.000,C 0.000} C_DIS
LIN {X 25.648,Y -288.864,Z 110.039,A 95.074,B 90.000,C 0.000} C_DIS
LIN {X 25.420,Y -288.884,Z 110.326,A 95.029,B 90.000,C 0.000} C_DIS
LIN {X 24.886,Y -288.930,Z 110.921,A 94.923,B 90.000,C 0.000} C_DIS
LIN {X 24.381,Y -288.973,Z 111.324,A 94.823,B 90.000,C 0.000} C_DIS
LIN {X 24.231,Y -288.986,Z 111.408,A 94.793,B 90.000,C 0.000} C_DIS
LIN {X 23.799,Y -289.022,Z 111.551,A 94.707,B 90.000,C 0.000} C_DIS
LIN {X 23.185,Y -289.072,Z 111.606,A 94.586,B 90.000,C 0.000} C_DIS
LIN {X 22.126,Y -289.155,Z 111.336,A 94.376,B 90.000,C 0.000} C_DIS
LIN {X 21.721,Y -289.185,Z 111.088,A 94.296,B 90.000,C 0.000} C_DIS
LIN {X 21.622,Y -289.193,Z 111.010,A 94.276,B 90.000,C 0.000} C_DIS
LIN {X 21.266,Y -289.219,Z 110.531,A 94.205,B 90.000,C 0.000} C_DIS
LIN {X 21.234,Y -289.222,Z 110.496,A 94.199,B 90.000,C 0.000} C_DIS
LIN {X 21.168,Y -289.226,Z 110.395,A 94.186,B 90.000,C 0.000} C_DIS
LIN {X 21.090,Y -289.232,Z 110.182,A 94.171,B 90.000,C 0.000} C_DIS
LIN {X 20.922,Y -289.244,Z 109.420,A 94.137,B 90.000,C 0.000} C_DIS
LIN {X 20.990,Y -289.239,Z 108.712,A 94.151,B 90.000,C 0.000} C_DIS
LIN {X 21.338,Y -289.214,Z 107.903,A 94.220,B 90.000,C 0.000} C_DIS
LIN {X 21.571,Y -289.197,Z 107.570,A 94.266,B 90.000,C 0.000} C_DIS
LIN {X 21.622,Y -289.193,Z 107.549,A 94.276,B 90.000,C 0.000} C_DIS
LIN {X 21.961,Y -289.167,Z 107.065,A 94.343,B 90.000,C 0.000} C_DIS
LIN {X 22.019,Y -289.163,Z 107.054,A 94.355,B 90.000,C 0.000} C_DIS
LIN {X 22.076,Y -289.159,Z 106.999,A 94.366,B 90.000,C 0.000} C_DIS
LIN {X 22.161,Y -289.152,Z 106.876,A 94.383,B 90.000,C 0.000} C_DIS
LIN {X 22.246,Y -289.145,Z 106.794,A 94.400,B 90.000,C 0.000} C_DIS
LIN {X 22.870,Y -289.097,Z 106.003,A 94.523,B 90.000,C 0.000} C_DIS
LIN {X 22.927,Y -289.092,Z 105.973,A 94.534,B 90.000,C 0.000} C_DIS
LIN {X 22.983,Y -289.088,Z 105.918,A 94.546,B 90.000,C 0.000} C_DIS
LIN {X 23.494,Y -289.047,Z 105.232,A 94.647,B 90.000,C 0.000} C_DIS
LIN {X 23.635,Y -289.035,Z 105.092,A 94.675,B 90.000,C 0.000} C_DIS
LIN {X 24.118,Y -288.995,Z 104.435,A 94.770,B 90.000,C 0.000} C_DIS
LIN {X 24.174,Y -288.991,Z 104.380,A 94.782,B 90.000,C 0.000} C_DIS
LIN {X 24.231,Y -288.986,Z 104.363,A 94.793,B 90.000,C 0.000} C_DIS
LIN {X 24.570,Y -288.957,Z 103.860,A 94.860,B 90.000,C 0.000} C_DIS
LIN {X 24.656,Y -288.950,Z 103.762,A 94.877,B 90.000,C 0.000} C_DIS
LIN {X 24.741,Y -288.943,Z 103.639,A 94.894,B 90.000,C 0.000} C_DIS
LIN {X 24.798,Y -288.938,Z 103.583,A 94.905,B 90.000,C 0.000} C_DIS
LIN {X 24.855,Y -288.933,Z 103.562,A 94.917,B 90.000,C 0.000} C_DIS
LIN {X 24.925,Y -288.927,Z 103.431,A 94.931,B 90.000,C 0.000} C_DIS
LIN {X 25.747,Y -288.855,Z 102.427,A 95.094,B 90.000,C 0.000} C_DIS
LIN {X 25.818,Y -288.848,Z 102.296,A 95.108,B 90.000,C 0.000} C_DIS
LIN {X 25.875,Y -288.843,Z 102.275,A 95.119,B 90.000,C 0.000} C_DIS
LIN {X 25.931,Y -288.838,Z 102.219,A 95.130,B 90.000,C 0.000} C_DIS
LIN {X 26.441,Y -288.792,Z 101.534,A 95.231,B 90.000,C 0.000} C_DIS
LIN {X 26.583,Y -288.779,Z 101.394,A 95.259,B 90.000,C 0.000} C_DIS
LIN {X 27.065,Y -288.734,Z 100.737,A 95.355,B 90.000,C 0.000} C_DIS
LIN {X 27.121,Y -288.729,Z 100.682,A 95.366,B 90.000,C 0.000} C_DIS
LIN {X 27.178,Y -288.724,Z 100.664,A 95.377,B 90.000,C 0.000} C_DIS
LIN {X 28.141,Y -288.631,Z 99.391,A 95.569,B 90.000,C 0.000} C_DIS
LIN {X 28.197,Y -288.626,Z 99.373,A 95.580,B 90.000,C 0.000} C_DIS
LIN {X 28.254,Y -288.620,Z 99.318,A 95.591,B 90.000,C 0.000} C_DIS
LIN {X 28.482,Y -288.598,Z 99.003,A 95.636,B 90.000,C 0.000} C_DIS
LIN {X 28.576,Y -288.589,Z 98.911,A 95.655,B 90.000,C 0.000} C_DIS
LIN {X 29.047,Y -288.542,Z 98.266,A 95.748,B 90.000,C 0.000} C_DIS
LIN {X 29.199,Y -288.526,Z 98.114,A 95.779,B 90.000,C 0.000} C_DIS
LIN {X 29.669,Y -288.478,Z 97.469,A 95.872,B 90.000,C 0.000} C_DIS
LIN {X 29.821,Y -288.463,Z 97.318,A 95.902,B 90.000,C 0.000} C_DIS
LIN {X 30.003,Y -288.444,Z 97.065,A 95.938,B 90.000,C 0.000} C_DIS
LIN {X 29.796,Y -286.454,Z 97.065,A 95.938,B 90.000,C 0.000} C_DIS
WAIT SEC 0.1
RET=EKI_SetBool("oxy","torchState",FALSE)
RET = EKI_Send("oxy","torchState")
LIN {X 27.934,Y -268.551,Z 97.065,A 95.938,B 90.000,C 0.000} C_DIS
LIN {X 34.520,Y -267.784,Z 100.539,A 97.346,B 90.000,C 0.000} C_DIS
LIN {X 36.822,Y -285.636,Z 100.539,A 97.346,B 90.000,C 0.000} C_DIS
LIN {X 37.077,Y -287.620,Z 100.539,A 97.346,B 90.000,C 0.000} C_DIS
WAIT SEC 1
RET=EKI_SetBool("oxy","torchState",TRUE)
RET = EKI_Send("oxy","torchState")
LIN {X 38.199,Y -287.473,Z 98.321,A 97.569,B 90.000,C 0.000} C_DIS
LIN {X 38.652,Y -287.413,Z 97.867,A 97.659,B 90.000,C 0.000} C_DIS
LIN {X 38.807,Y -287.392,Z 97.663,A 97.690,B 90.000,C 0.000} C_DIS
LIN {X 38.878,Y -287.382,Z 97.526,A 97.704,B 90.000,C 0.000} C_DIS
LIN {X 39.372,Y -287.315,Z 96.862,A 97.803,B 90.000,C 0.000} C_DIS
LIN {X 39.780,Y -287.259,Z 96.513,A 97.884,B 90.000,C 0.000} C_DIS
LIN {X 39.935,Y -287.237,Z 96.427,A 97.915,B 90.000,C 0.000} C_DIS
LIN {X 40.442,Y -287.166,Z 96.439,A 98.016,B 90.000,C 0.000} C_DIS
LIN {X 40.829,Y -287.111,Z 96.727,A 98.094,B 90.000,C 0.000} C_DIS
LIN {X 41.254,Y -287.051,Z 97.638,A 98.178,B 90.000,C 0.000} C_DIS
LIN {X 41.298,Y -287.044,Z 97.752,A 98.187,B 90.000,C 0.000} C_DIS
LIN {X 41.417,Y -287.027,Z 97.922,A 98.211,B 90.000,C 0.000} C_DIS
LIN {X 41.467,Y -287.020,Z 98.036,A 98.221,B 90.000,C 0.000} C_DIS
LIN {X 41.808,Y -286.971,Z 98.524,A 98.289,B 90.000,C 0.000} C_DIS
LIN {X 42.033,Y -286.938,Z 98.893,A 98.334,B 90.000,C 0.000} C_DIS
LIN {X 42.538,Y -286.863,Z 99.502,A 98.435,B 90.000,C 0.000} C_DIS
LIN {X 42.796,Y -286.825,Z 99.904,A 98.486,B 90.000,C 0.000} C_DIS
LIN {X 42.949,Y -286.802,Z 100.084,A 98.517,B 90.000,C 0.000} C_DIS
LIN {X 42.962,Y -286.800,Z 100.141,A 98.519,B 90.000,C 0.000} C_DIS
LIN {X 42.986,Y -286.796,Z 100.198,A 98.524,B 90.000,C 0.000} C_DIS
LIN {X 43.046,Y -286.787,Z 100.283,A 98.536,B 90.000,C 0.000} C_DIS
LIN {X 43.089,Y -286.781,Z 100.369,A 98.545,B 90.000,C 0.000} C_DIS
LIN {X 43.453,Y -286.726,Z 100.881,A 98.617,B 90.000,C 0.000} C_DIS
LIN {X 43.570,Y -286.708,Z 101.119,A 98.641,B 90.000,C 0.000} C_DIS
LIN {X 43.905,Y -286.657,Z 101.564,A 98.708,B 90.000,C 0.000} C_DIS
LIN {X 43.918,Y -286.655,Z 101.621,A 98.710,B 90.000,C 0.000} C_DIS
LIN {X 43.943,Y -286.651,Z 101.677,A 98.715,B 90.000,C 0.000} C_DIS
LIN {X 44.002,Y -286.642,Z 101.738,A 98.727,B 90.000,C 0.000} C_DIS
LIN {X 44.073,Y -286.631,Z 101.879,A 98.741,B 90.000,C 0.000} C_DIS
LIN {X 44.743,Y -286.528,Z 102.648,A 98.875,B 90.000,C 0.000} C_DIS
LIN {X 45.252,Y -286.448,Z 103.327,A 98.977,B 90.000,C 0.000} C_DIS
LIN {X 45.295,Y -286.441,Z 103.413,A 98.986,B 90.000,C 0.000} C_DIS
LIN {X 45.355,Y -286.431,Z 103.498,A 98.998,B 90.000,C 0.000} C_DIS
LIN {X 45.380,Y -286.427,Z 103.555,A 99.003,B 90.000,C 0.000} C_DIS
LIN {X 45.392,Y -286.425,Z 103.612,A 99.005,B 90.000,C 0.000} C_DIS
LIN {X 46.307,Y -286.279,Z 104.693,A 99.188,B 90.000,C 0.000} C_DIS
LIN {X 46.381,Y -286.267,Z 104.750,A 99.203,B 90.000,C 0.000} C_DIS
LIN {X 46.653,Y -286.223,Z 105.034,A 99.258,B 90.000,C 0.000} C_DIS
LIN {X 48.327,Y -285.945,Z 106.458,A 99.593,B 90.000,C 0.000} C_DIS
LIN {X 48.424,Y -285.928,Z 106.555,A 99.612,B 90.000,C 0.000} C_DIS
LIN {X 48.846,Y -285.857,Z 106.872,A 99.697,B 90.000,C 0.000} C_DIS
LIN {X 49.004,Y -285.830,Z 107.026,A 99.729,B 90.000,C 0.000} C_DIS
LIN {X 49.138,Y -285.807,Z 107.097,A 99.755,B 90.000,C 0.000} C_DIS
LIN {X 49.575,Y -285.731,Z 107.438,A 99.843,B 90.000,C 0.000} C_DIS
LIN {X 49.769,Y -285.697,Z 107.538,A 99.882,B 90.000,C 0.000} C_DIS
LIN {X 49.813,Y -285.690,Z 107.595,A 99.891,B 90.000,C 0.000} C_DIS
LIN {X 49.829,Y -285.687,Z 107.651,A 99.894,B 90.000,C 0.000} C_DIS
LIN {X 50.217,Y -285.619,Z 107.935,A 99.972,B 90.000,C 0.000} C_DIS
LIN {X 50.337,Y -285.598,Z 107.993,A 99.996,B 90.000,C 0.000} C_DIS
LIN {X 50.422,Y -285.583,Z 108.078,A 100.013,B 90.000,C 0.000} C_DIS
LIN {X 50.626,Y -285.547,Z 108.217,A 100.054,B 90.000,C 0.000} C_DIS
LIN {X 50.739,Y -285.527,Z 108.306,A 100.076,B 90.000,C 0.000} C_DIS
LIN {X 50.876,Y -285.502,Z 108.448,A 100.104,B 90.000,C 0.000} C_DIS
LIN {X 50.998,Y -285.481,Z 108.533,A 100.128,B 90.000,C 0.000} C_DIS
LIN {X 51.094,Y -285.463,Z 108.620,A 100.148,B 90.000,C 0.000} C_DIS
LIN {X 51.608,Y -285.371,Z 108.960,A 100.251,B 90.000,C 0.000} C_DIS
LIN {X 51.914,Y -285.316,Z 109.184,A 100.312,B 90.000,C 0.000} C_DIS
LIN {X 52.027,Y -285.295,Z 109.273,A 100.335,B 90.000,C 0.000} C_DIS
LIN {X 52.164,Y -285.270,Z 109.415,A 100.363,B 90.000,C 0.000} C_DIS
LIN {X 52.529,Y -285.203,Z 109.644,A 100.436,B 90.000,C 0.000} C_DIS
LIN {X 52.869,Y -285.140,Z 109.927,A 100.504,B 90.000,C 0.000} C_DIS
LIN {X 53.002,Y -285.115,Z 109.998,A 100.531,B 90.000,C 0.000} C_DIS
LIN {X 53.399,Y -285.041,Z 110.311,A 100.611,B 90.000,C 0.000} C_DIS
LIN {X 53.524,Y -285.018,Z 110.382,A 100.636,B 90.000,C 0.000} C_DIS
LIN {X 53.911,Y -284.945,Z 110.666,A 100.714,B 90.000,C 0.000} C_DIS
LIN {X 54.031,Y -284.922,Z 110.724,A 100.738,B 90.000,C 0.000} C_DIS
LIN {X 54.116,Y -284.906,Z 110.809,A 100.755,B 90.000,C 0.000} C_DIS
LIN {X 54.598,Y -284.814,Z 111.130,A 100.852,B 90.000,C 0.000} C_DIS
LIN {X 55.555,Y -284.629,Z 111.862,A 101.044,B 90.000,C 0.000} C_DIS
LIN {X 55.728,Y -284.595,Z 112.146,A 101.079,B 90.000,C 0.000} C_DIS
LIN {X 55.781,Y -284.585,Z 112.374,A 101.090,B 90.000,C 0.000} C_DIS
LIN {X 55.800,Y -284.581,Z 112.543,A 101.094,B 90.000,C 0.000} C_DIS
LIN {X 55.643,Y -284.612,Z 115.037,A 101.062,B 90.000,C 0.000} C_DIS
LIN {X 55.600,Y -284.620,Z 115.794,A 101.053,B 90.000,C 0.000} C_DIS
LIN {X 55.458,Y -284.648,Z 116.248,A 101.025,B 90.000,C 0.000} C_DIS
LIN {X 55.380,Y -284.663,Z 116.418,A 101.009,B 90.000,C 0.000} C_DIS
LIN {X 55.245,Y -284.689,Z 116.581,A 100.982,B 90.000,C 0.000} C_DIS
LIN {X 52.789,Y -285.151,Z 116.627,A 100.488,B 90.000,C 0.000} C_DIS
LIN {X 51.526,Y -285.386,Z 116.615,A 100.234,B 90.000,C 0.000} C_DIS
LIN {X 51.407,Y -285.407,Z 116.668,A 100.211,B 90.000,C 0.000} C_DIS
LIN {X 49.603,Y -285.726,Z 116.556,A 99.849,B 90.000,C 0.000} C_DIS
LIN {X 49.505,Y -285.743,Z 116.581,A 99.829,B 90.000,C 0.000} C_DIS
LIN {X 49.453,Y -285.752,Z 116.615,A 99.819,B 90.000,C 0.000} C_DIS
LIN {X 48.173,Y -285.971,Z 116.504,A 99.562,B 90.000,C 0.000} C_DIS
LIN {X 48.047,Y -285.992,Z 116.524,A 99.537,B 90.000,C 0.000} C_DIS
LIN {X 45.599,Y -286.392,Z 116.212,A 99.047,B 90.000,C 0.000} C_DIS
LIN {X 44.227,Y -286.608,Z 116.077,A 98.772,B 90.000,C 0.000} C_DIS
LIN {X 44.101,Y -286.627,Z 116.099,A 98.747,B 90.000,C 0.000} C_DIS
LIN {X 41.665,Y -286.991,Z 115.671,A 98.260,B 90.000,C 0.000} C_DIS
LIN {X 39.267,Y -287.329,Z 115.049,A 97.782,B 90.000,C 0.000} C_DIS
LIN {X 36.893,Y -287.644,Z 114.333,A 97.309,B 90.000,C 0.000} C_DIS
LIN {X 34.516,Y -287.939,Z 113.616,A 96.836,B 90.000,C 0.000} C_DIS
LIN {X 33.735,Y -288.031,Z 113.284,A 96.680,B 90.000,C 0.000} C_DIS
LIN {X 33.592,Y -288.048,Z 113.199,A 96.652,B 90.000,C 0.000} C_DIS
LIN {X 33.478,Y -288.061,Z 113.113,A 96.629,B 90.000,C 0.000} C_DIS
LIN {X 33.329,Y -288.078,Z 113.058,A 96.599,B 90.000,C 0.000} C_DIS
LIN {X 32.939,Y -288.123,Z 112.740,A 96.522,B 90.000,C 0.000} C_DIS
LIN {X 33.289,Y -288.083,Z 111.046,A 96.592,B 90.000,C 0.000} C_DIS
LIN {X 33.336,Y -288.078,Z 111.031,A 96.601,B 90.000,C 0.000} C_DIS
LIN {X 34.141,Y -287.983,Z 108.666,A 96.761,B 90.000,C 0.000} C_DIS
LIN {X 34.983,Y -287.882,Z 106.314,A 96.929,B 90.000,C 0.000} C_DIS
LIN {X 35.762,Y -287.787,Z 103.941,A 97.084,B 90.000,C 0.000} C_DIS
LIN {X 36.614,Y -287.679,Z 101.593,A 97.253,B 90.000,C 0.000} C_DIS
LIN {X 37.077,Y -287.620,Z 100.539,A 97.346,B 90.000,C 0.000} C_DIS
LIN {X 36.822,Y -285.636,Z 100.539,A 97.346,B 90.000,C 0.000} C_DIS
WAIT SEC 0.1
RET=EKI_SetBool("oxy","torchState",FALSE)
RET = EKI_Send("oxy","torchState")
LIN {X 34.520,Y -267.784,Z 100.539,A 97.346,B 90.000,C 0.000} C_DIS
LIN {X 37.009,Y -267.452,Z 89.089,A 97.878,B 90.000,C 0.000} C_DIS
LIN {X 39.476,Y -285.282,Z 89.089,A 97.878,B 90.000,C 0.000} C_DIS
LIN {X 39.750,Y -287.263,Z 89.089,A 97.878,B 90.000,C 0.000} C_DIS
WAIT SEC 1
RET=EKI_SetBool("oxy","torchState",TRUE)
RET = EKI_Send("oxy","torchState")
LIN {X 40.974,Y -287.091,Z 89.258,A 98.122,B 90.000,C 0.000} C_DIS
LIN {X 41.723,Y -286.983,Z 89.104,A 98.272,B 90.000,C 0.000} C_DIS
LIN {X 42.053,Y -286.935,Z 88.961,A 98.338,B 90.000,C 0.000} C_DIS
LIN {X 42.597,Y -286.854,Z 88.573,A 98.447,B 90.000,C 0.000} C_DIS
LIN {X 43.018,Y -286.792,Z 88.116,A 98.531,B 90.000,C 0.000} C_DIS
LIN {X 43.102,Y -286.779,Z 88.000,A 98.547,B 90.000,C 0.000} C_DIS
LIN {X 43.320,Y -286.746,Z 87.508,A 98.591,B 90.000,C 0.000} C_DIS
LIN {X 43.470,Y -286.724,Z 86.818,A 98.621,B 90.000,C 0.000} C_DIS
LIN {X 43.475,Y -286.723,Z 85.966,A 98.622,B 90.000,C 0.000} C_DIS
LIN {X 43.290,Y -286.751,Z 85.359,A 98.585,B 90.000,C 0.000} C_DIS
LIN {X 43.215,Y -286.762,Z 85.200,A 98.570,B 90.000,C 0.000} C_DIS
LIN {X 42.845,Y -286.818,Z 84.634,A 98.496,B 90.000,C 0.000} C_DIS
LIN {X 42.172,Y -286.917,Z 84.070,A 98.362,B 90.000,C 0.000} C_DIS
LIN {X 41.842,Y -286.966,Z 83.875,A 98.296,B 90.000,C 0.000} C_DIS
LIN {X 40.858,Y -287.107,Z 83.648,A 98.099,B 90.000,C 0.000} C_DIS
LIN {X 39.611,Y -287.282,Z 83.954,A 97.850,B 90.000,C 0.000} C_DIS
LIN {X 39.554,Y -287.290,Z 83.979,A 97.839,B 90.000,C 0.000} C_DIS
LIN {X 39.468,Y -287.302,Z 84.040,A 97.822,B 90.000,C 0.000} C_DIS
LIN {X 39.173,Y -287.342,Z 84.192,A 97.763,B 90.000,C 0.000} C_DIS
LIN {X 38.769,Y -287.397,Z 84.547,A 97.683,B 90.000,C 0.000} C_DIS
LIN {X 38.411,Y -287.445,Z 84.949,A 97.611,B 90.000,C 0.000} C_DIS
LIN {X 38.181,Y -287.476,Z 85.401,A 97.565,B 90.000,C 0.000} C_DIS
LIN {X 37.964,Y -287.504,Z 86.272,A 97.522,B 90.000,C 0.000} C_DIS
LIN {X 37.925,Y -287.509,Z 86.776,A 97.514,B 90.000,C 0.000} C_DIS
LIN {X 37.992,Y -287.501,Z 87.112,A 97.528,B 90.000,C 0.000} C_DIS
LIN {X 38.072,Y -287.490,Z 87.340,A 97.544,B 90.000,C 0.000} C_DIS
LIN {X 38.088,Y -287.488,Z 87.453,A 97.547,B 90.000,C 0.000} C_DIS
LIN {X 38.210,Y -287.472,Z 87.809,A 97.571,B 90.000,C 0.000} C_DIS
LIN {X 38.254,Y -287.466,Z 87.852,A 97.580,B 90.000,C 0.000} C_DIS
LIN {X 38.714,Y -287.404,Z 88.414,A 97.672,B 90.000,C 0.000} C_DIS
LIN {X 39.296,Y -287.325,Z 88.876,A 97.788,B 90.000,C 0.000} C_DIS
LIN {X 39.425,Y -287.308,Z 88.955,A 97.813,B 90.000,C 0.000} C_DIS
LIN {X 39.750,Y -287.263,Z 89.089,A 97.878,B 90.000,C 0.000} C_DIS
LIN {X 39.476,Y -285.282,Z 89.089,A 97.878,B 90.000,C 0.000} C_DIS
WAIT SEC 0.1
RET=EKI_SetBool("oxy","torchState",FALSE)
RET = EKI_Send("oxy","torchState")
LIN {X 37.009,Y -267.452,Z 89.089,A 97.878,B 90.000,C 0.000} C_DIS
LIN {X 42.030,Y -266.709,Z 87.567,A 98.955,B 90.000,C 0.000} C_DIS
LIN {X 44.832,Y -284.489,Z 87.567,A 98.955,B 90.000,C 0.000} C_DIS
LIN {X 45.143,Y -286.465,Z 87.567,A 98.955,B 90.000,C 0.000} C_DIS
WAIT SEC 1
RET=EKI_SetBool("oxy","torchState",TRUE)
RET = EKI_Send("oxy","torchState")
LIN {X 45.011,Y -286.486,Z 86.828,A 98.929,B 90.000,C 0.000} C_DIS
LIN {X 44.966,Y -286.493,Z 86.589,A 98.920,B 90.000,C 0.000} C_DIS
LIN {X 45.108,Y -286.470,Z 85.521,A 98.948,B 90.000,C 0.000} C_DIS
LIN {X 45.221,Y -286.453,Z 85.251,A 98.971,B 90.000,C 0.000} C_DIS
LIN {X 45.295,Y -286.441,Z 85.143,A 98.986,B 90.000,C 0.000} C_DIS
LIN {X 45.337,Y -286.434,Z 85.064,A 98.994,B 90.000,C 0.000} C_DIS
LIN {X 45.543,Y -286.402,Z 84.921,A 99.035,B 90.000,C 0.000} C_DIS
LIN {X 45.942,Y -286.338,Z 84.721,A 99.115,B 90.000,C 0.000} C_DIS
LIN {X 46.030,Y -286.324,Z 84.696,A 99.133,B 90.000,C 0.000} C_DIS
LIN {X 46.082,Y -286.315,Z 84.662,A 99.143,B 90.000,C 0.000} C_DIS
LIN {X 46.250,Y -286.288,Z 84.628,A 99.177,B 90.000,C 0.000} C_DIS
LIN {X 48.716,Y -285.878,Z 84.652,A 99.671,B 90.000,C 0.000} C_DIS
LIN {X 49.448,Y -285.753,Z 84.693,A 99.817,B 90.000,C 0.000} C_DIS
LIN {X 49.505,Y -285.743,Z 84.669,A 99.829,B 90.000,C 0.000} C_DIS
LIN {X 49.592,Y -285.728,Z 84.611,A 99.846,B 90.000,C 0.000} C_DIS
LIN {X 49.721,Y -285.706,Z 84.708,A 99.872,B 90.000,C 0.000} C_DIS
LIN {X 49.709,Y -285.708,Z 87.208,A 99.870,B 90.000,C 0.000} C_DIS
LIN {X 49.706,Y -285.708,Z 87.730,A 99.869,B 90.000,C 0.000} C_DIS
LIN {X 49.730,Y -285.704,Z 87.795,A 99.874,B 90.000,C 0.000} C_DIS
LIN {X 49.752,Y -285.700,Z 87.923,A 99.879,B 90.000,C 0.000} C_DIS
LIN {X 49.654,Y -285.717,Z 90.421,A 99.859,B 90.000,C 0.000} C_DIS
LIN {X 49.585,Y -285.729,Z 92.920,A 99.845,B 90.000,C 0.000} C_DIS
LIN {X 49.496,Y -285.745,Z 95.418,A 99.827,B 90.000,C 0.000} C_DIS
LIN {X 49.480,Y -285.748,Z 95.698,A 99.824,B 90.000,C 0.000} C_DIS
LIN {X 49.497,Y -285.745,Z 95.760,A 99.827,B 90.000,C 0.000} C_DIS
LIN {X 49.519,Y -285.741,Z 95.945,A 99.832,B 90.000,C 0.000} C_DIS
LIN {X 49.483,Y -285.747,Z 96.343,A 99.825,B 90.000,C 0.000} C_DIS
LIN {X 49.408,Y -285.760,Z 96.557,A 99.810,B 90.000,C 0.000} C_DIS
LIN {X 49.337,Y -285.772,Z 96.471,A 99.795,B 90.000,C 0.000} C_DIS
LIN {X 49.106,Y -285.812,Z 96.102,A 99.749,B 90.000,C 0.000} C_DIS
LIN {X 48.980,Y -285.834,Z 95.804,A 99.724,B 90.000,C 0.000} C_DIS
LIN {X 48.249,Y -285.958,Z 94.385,A 99.577,B 90.000,C 0.000} C_DIS
LIN {X 48.100,Y -285.983,Z 94.167,A 99.547,B 90.000,C 0.000} C_DIS
LIN {X 48.072,Y -285.988,Z 94.115,A 99.542,B 90.000,C 0.000} C_DIS
LIN {X 48.061,Y -285.990,Z 94.044,A 99.540,B 90.000,C 0.000} C_DIS
LIN {X 47.597,Y -286.067,Z 93.100,A 99.446,B 90.000,C 0.000} C_DIS
LIN {X 46.531,Y -286.243,Z 91.005,A 99.233,B 90.000,C 0.000} C_DIS
LIN {X 46.478,Y -286.251,Z 90.924,A 99.223,B 90.000,C 0.000} C_DIS
LIN {X 46.417,Y -286.261,Z 90.696,A 99.210,B 90.000,C 0.000} C_DIS
LIN {X 46.194,Y -286.297,Z 90.311,A 99.166,B 90.000,C 0.000} C_DIS
LIN {X 45.675,Y -286.380,Z 88.975,A 99.062,B 90.000,C 0.000} C_DIS
LIN {X 45.635,Y -286.387,Z 88.933,A 99.054,B 90.000,C 0.000} C_DIS
LIN {X 45.235,Y -286.450,Z 87.909,A 98.974,B 90.000,C 0.000} C_DIS
LIN {X 45.223,Y -286.452,Z 87.795,A 98.971,B 90.000,C 0.000} C_DIS
LIN {X 45.143,Y -286.465,Z 87.567,A 98.955,B 90.000,C 0.000} C_DIS
LIN {X 44.832,Y -284.489,Z 87.567,A 98.955,B 90.000,C 0.000} C_DIS
WAIT SEC 0.1
RET=EKI_SetBool("oxy","torchState",FALSE)
RET = EKI_Send("oxy","torchState")
LIN {X 42.030,Y -266.709,Z 87.567,A 98.955,B 90.000,C 0.000} C_DIS
LIN {X 48.881,Y -265.538,Z 88.506,A 100.430,B 90.000,C 0.000} C_DIS
LIN {X 52.139,Y -283.241,Z 88.506,A 100.430,B 90.000,C 0.000} C_DIS
LIN {X 52.501,Y -285.208,Z 88.506,A 100.430,B 90.000,C 0.000} C_DIS
WAIT SEC 1
RET=EKI_SetBool("oxy","torchState",TRUE)
RET = EKI_Send("oxy","torchState")
LIN {X 52.425,Y -285.222,Z 91.005,A 100.415,B 90.000,C 0.000} C_DIS
LIN {X 52.357,Y -285.235,Z 93.504,A 100.401,B 90.000,C 0.000} C_DIS
LIN {X 52.292,Y -285.247,Z 96.003,A 100.388,B 90.000,C 0.000} C_DIS
LIN {X 52.222,Y -285.259,Z 97.424,A 100.374,B 90.000,C 0.000} C_DIS
LIN {X 52.247,Y -285.255,Z 97.581,A 100.379,B 90.000,C 0.000} C_DIS
LIN {X 52.276,Y -285.249,Z 97.640,A 100.385,B 90.000,C 0.000} C_DIS
LIN {X 52.168,Y -285.269,Z 99.455,A 100.363,B 90.000,C 0.000} C_DIS
LIN {X 52.218,Y -285.260,Z 99.634,A 100.373,B 90.000,C 0.000} C_DIS
LIN {X 52.061,Y -285.289,Z 101.720,A 100.342,B 90.000,C 0.000} C_DIS
LIN {X 52.178,Y -285.267,Z 102.468,A 100.365,B 90.000,C 0.000} C_DIS
LIN {X 53.216,Y -285.076,Z 104.260,A 100.574,B 90.000,C 0.000} C_DIS
LIN {X 53.313,Y -285.057,Z 104.367,A 100.593,B 90.000,C 0.000} C_DIS
LIN {X 53.533,Y -285.016,Z 104.693,A 100.638,B 90.000,C 0.000} C_DIS
LIN {X 53.889,Y -284.949,Z 105.055,A 100.709,B 90.000,C 0.000} C_DIS
LIN {X 54.312,Y -284.869,Z 105.198,A 100.794,B 90.000,C 0.000} C_DIS
LIN {X 55.919,Y -284.558,Z 105.212,A 101.118,B 90.000,C 0.000} C_DIS
LIN {X 56.077,Y -284.527,Z 105.178,A 101.149,B 90.000,C 0.000} C_DIS
LIN {X 56.172,Y -284.508,Z 105.050,A 101.169,B 90.000,C 0.000} C_DIS
LIN {X 56.326,Y -284.477,Z 102.555,A 101.200,B 90.000,C 0.000} C_DIS
LIN {X 56.424,Y -284.458,Z 100.058,A 101.219,B 90.000,C 0.000} C_DIS
LIN {X 56.507,Y -284.442,Z 97.559,A 101.236,B 90.000,C 0.000} C_DIS
LIN {X 56.579,Y -284.427,Z 95.060,A 101.251,B 90.000,C 0.000} C_DIS
LIN {X 56.632,Y -284.417,Z 94.067,A 101.261,B 90.000,C 0.000} C_DIS
LIN {X 56.609,Y -284.421,Z 93.940,A 101.257,B 90.000,C 0.000} C_DIS
LIN {X 56.584,Y -284.426,Z 93.877,A 101.252,B 90.000,C 0.000} C_DIS
LIN {X 56.672,Y -284.409,Z 91.379,A 101.269,B 90.000,C 0.000} C_DIS
LIN {X 56.720,Y -284.399,Z 88.879,A 101.279,B 90.000,C 0.000} C_DIS
LIN {X 56.799,Y -284.383,Z 86.389,A 101.295,B 90.000,C 0.000} C_DIS
LIN {X 56.777,Y -284.388,Z 86.231,A 101.291,B 90.000,C 0.000} C_DIS
LIN {X 56.748,Y -284.394,Z 86.145,A 101.285,B 90.000,C 0.000} C_DIS
LIN {X 56.812,Y -284.381,Z 85.119,A 101.298,B 90.000,C 0.000} C_DIS
LIN {X 56.658,Y -284.412,Z 84.924,A 101.266,B 90.000,C 0.000} C_DIS
LIN {X 54.209,Y -284.888,Z 84.762,A 100.774,B 90.000,C 0.000} C_DIS
LIN {X 54.100,Y -284.909,Z 84.754,A 100.752,B 90.000,C 0.000} C_DIS
LIN {X 54.039,Y -284.921,Z 84.770,A 100.739,B 90.000,C 0.000} C_DIS
LIN {X 53.550,Y -285.013,Z 84.749,A 100.641,B 90.000,C 0.000} C_DIS
LIN {X 53.480,Y -285.026,Z 84.775,A 100.627,B 90.000,C 0.000} C_DIS
LIN {X 52.991,Y -285.117,Z 84.749,A 100.529,B 90.000,C 0.000} C_DIS
LIN {X 52.921,Y -285.130,Z 84.788,A 100.515,B 90.000,C 0.000} C_DIS
LIN {X 52.809,Y -285.151,Z 84.820,A 100.492,B 90.000,C 0.000} C_DIS
LIN {X 52.717,Y -285.168,Z 84.811,A 100.474,B 90.000,C 0.000} C_DIS
LIN {X 52.665,Y -285.178,Z 84.880,A 100.463,B 90.000,C 0.000} C_DIS
LIN {X 52.556,Y -285.198,Z 86.089,A 100.441,B 90.000,C 0.000} C_DIS
LIN {X 52.586,Y -285.192,Z 86.145,A 100.447,B 90.000,C 0.000} C_DIS
LIN {X 52.610,Y -285.188,Z 86.270,A 100.452,B 90.000,C 0.000} C_DIS
LIN {X 52.501,Y -285.208,Z 88.506,A 100.430,B 90.000,C 0.000} C_DIS
LIN {X 52.139,Y -283.241,Z 88.506,A 100.430,B 90.000,C 0.000} C_DIS
WAIT SEC 0.1
RET=EKI_SetBool("oxy","torchState",FALSE)
RET = EKI_Send("oxy","torchState")
LIN {X 48.881,Y -265.538,Z 88.506,A 100.430,B 90.000,C 0.000} C_DIS
LIN {X 55.384,Y -264.259,Z 89.022,A 101.837,B 90.000,C 0.000} C_DIS
LIN {X 59.076,Y -281.876,Z 89.022,A 101.837,B 90.000,C 0.000} C_DIS
LIN {X 59.486,Y -283.833,Z 89.022,A 101.837,B 90.000,C 0.000} C_DIS
WAIT SEC 1
RET=EKI_SetBool("oxy","torchState",TRUE)
RET = EKI_Send("oxy","torchState")
LIN {X 59.587,Y -283.812,Z 86.668,A 101.857,B 90.000,C 0.000} C_DIS
LIN {X 59.607,Y -283.808,Z 85.178,A 101.861,B 90.000,C 0.000} C_DIS
LIN {X 59.549,Y -283.820,Z 85.154,A 101.849,B 90.000,C 0.000} C_DIS
LIN {X 59.585,Y -283.813,Z 85.101,A 101.857,B 90.000,C 0.000} C_DIS
LIN {X 59.818,Y -283.764,Z 85.003,A 101.904,B 90.000,C 0.000} C_DIS
LIN {X 61.787,Y -283.341,Z 85.034,A 102.302,B 90.000,C 0.000} C_DIS
LIN {X 61.844,Y -283.329,Z 85.018,A 102.313,B 90.000,C 0.000} C_DIS
LIN {X 63.229,Y -283.023,Z 85.023,A 102.593,B 90.000,C 0.000} C_DIS
LIN {X 63.432,Y -282.978,Z 85.130,A 102.635,B 90.000,C 0.000} C_DIS
LIN {X 63.485,Y -282.966,Z 85.520,A 102.645,B 90.000,C 0.000} C_DIS
LIN {X 63.433,Y -282.977,Z 88.020,A 102.635,B 90.000,C 0.000} C_DIS
LIN {X 63.372,Y -282.991,Z 90.519,A 102.622,B 90.000,C 0.000} C_DIS
LIN {X 63.323,Y -283.002,Z 92.560,A 102.612,B 90.000,C 0.000} C_DIS
LIN {X 63.368,Y -282.992,Z 92.751,A 102.622,B 90.000,C 0.000} C_DIS
LIN {X 63.258,Y -283.017,Z 95.248,A 102.599,B 90.000,C 0.000} C_DIS
LIN {X 63.210,Y -283.027,Z 96.549,A 102.590,B 90.000,C 0.000} C_DIS
LIN {X 63.234,Y -283.022,Z 96.614,A 102.594,B 90.000,C 0.000} C_DIS
LIN {X 63.258,Y -283.017,Z 96.737,A 102.599,B 90.000,C 0.000} C_DIS
LIN {X 63.152,Y -283.040,Z 98.544,A 102.578,B 90.000,C 0.000} C_DIS
LIN {X 63.205,Y -283.029,Z 98.663,A 102.588,B 90.000,C 0.000} C_DIS
LIN {X 63.100,Y -283.052,Z 101.161,A 102.567,B 90.000,C 0.000} C_DIS
LIN {X 63.046,Y -283.064,Z 101.950,A 102.556,B 90.000,C 0.000} C_DIS
LIN {X 63.088,Y -283.055,Z 102.143,A 102.565,B 90.000,C 0.000} C_DIS
LIN {X 62.975,Y -283.080,Z 104.640,A 102.542,B 90.000,C 0.000} C_DIS
LIN {X 62.963,Y -283.082,Z 104.988,A 102.540,B 90.000,C 0.000} C_DIS
LIN {X 62.877,Y -283.101,Z 105.350,A 102.522,B 90.000,C 0.000} C_DIS
LIN {X 60.434,Y -283.632,Z 105.359,A 102.028,B 90.000,C 0.000} C_DIS
LIN {X 59.179,Y -283.898,Z 105.294,A 101.775,B 90.000,C 0.000} C_DIS
LIN {X 59.101,Y -283.914,Z 104.994,A 101.759,B 90.000,C 0.000} C_DIS
LIN {X 59.108,Y -283.912,Z 103.065,A 101.760,B 90.000,C 0.000} C_DIS
LIN {X 59.095,Y -283.915,Z 102.978,A 101.758,B 90.000,C 0.000} C_DIS
LIN {X 59.170,Y -283.899,Z 100.479,A 101.773,B 90.000,C 0.000} C_DIS
LIN {X 59.200,Y -283.893,Z 99.501,A 101.779,B 90.000,C 0.000} C_DIS
LIN {X 59.176,Y -283.898,Z 99.345,A 101.774,B 90.000,C 0.000} C_DIS
LIN {X 59.149,Y -283.904,Z 99.282,A 101.769,B 90.000,C 0.000} C_DIS
LIN {X 59.255,Y -283.882,Z 96.785,A 101.790,B 90.000,C 0.000} C_DIS
LIN {X 59.338,Y -283.864,Z 94.286,A 101.807,B 90.000,C 0.000} C_DIS
LIN {X 59.367,Y -283.858,Z 93.430,A 101.813,B 90.000,C 0.000} C_DIS
LIN {X 59.317,Y -283.869,Z 93.306,A 101.803,B 90.000,C 0.000} C_DIS
LIN {X 59.444,Y -283.842,Z 90.810,A 101.828,B 90.000,C 0.000} C_DIS
LIN {X 59.475,Y -283.836,Z 90.078,A 101.835,B 90.000,C 0.000} C_DIS
LIN {X 59.451,Y -283.841,Z 90.014,A 101.830,B 90.000,C 0.000} C_DIS
LIN {X 59.427,Y -283.846,Z 89.890,A 101.825,B 90.000,C 0.000} C_DIS
LIN {X 59.486,Y -283.833,Z 89.022,A 101.837,B 90.000,C 0.000} C_DIS
LIN {X 59.076,Y -281.876,Z 89.022,A 101.837,B 90.000,C 0.000} C_DIS
WAIT SEC 0.1
RET=EKI_SetBool("oxy","torchState",FALSE)
RET = EKI_Send("oxy","torchState")
LIN {X 55.384,Y -264.259,Z 89.022,A 101.837,B 90.000,C 0.000} C_DIS
LIN {X 61.732,Y -262.848,Z 88.727,A 103.217,B 90.000,C 0.000} C_DIS
LIN {X 65.847,Y -280.372,Z 88.727,A 103.217,B 90.000,C 0.000} C_DIS
LIN {X 66.304,Y -282.319,Z 88.727,A 103.217,B 90.000,C 0.000} C_DIS
WAIT SEC 1
RET=EKI_SetBool("oxy","torchState",TRUE)
RET = EKI_Send("oxy","torchState")
LIN {X 66.362,Y -282.305,Z 87.916,A 103.228,B 90.000,C 0.000} C_DIS
LIN {X 66.339,Y -282.310,Z 87.852,A 103.224,B 90.000,C 0.000} C_DIS
LIN {X 66.311,Y -282.317,Z 87.795,A 103.218,B 90.000,C 0.000} C_DIS
LIN {X 66.438,Y -282.287,Z 85.298,A 103.244,B 90.000,C 0.000} C_DIS
LIN {X 66.449,Y -282.284,Z 85.137,A 103.246,B 90.000,C 0.000} C_DIS
LIN {X 67.558,Y -282.021,Z 85.206,A 103.471,B 90.000,C 0.000} C_DIS
LIN {X 67.723,Y -281.982,Z 85.179,A 103.505,B 90.000,C 0.000} C_DIS
LIN {X 67.777,Y -281.968,Z 85.149,A 103.516,B 90.000,C 0.000} C_DIS
LIN {X 70.200,Y -281.375,Z 85.315,A 104.009,B 90.000,C 0.000} C_DIS
LIN {X 70.254,Y -281.362,Z 85.319,A 104.020,B 90.000,C 0.000} C_DIS
LIN {X 70.246,Y -281.364,Z 86.671,A 104.018,B 90.000,C 0.000} C_DIS
LIN {X 70.272,Y -281.357,Z 86.828,A 104.023,B 90.000,C 0.000} C_DIS
LIN {X 70.289,Y -281.353,Z 86.889,A 104.027,B 90.000,C 0.000} C_DIS
LIN {X 70.211,Y -281.372,Z 89.388,A 104.011,B 90.000,C 0.000} C_DIS
LIN {X 70.132,Y -281.392,Z 91.825,A 103.995,B 90.000,C 0.000} C_DIS
LIN {X 70.157,Y -281.386,Z 91.891,A 104.000,B 90.000,C 0.000} C_DIS
LIN {X 70.182,Y -281.380,Z 91.991,A 104.005,B 90.000,C 0.000} C_DIS
LIN {X 70.074,Y -281.407,Z 94.391,A 103.983,B 90.000,C 0.000} C_DIS
LIN {X 70.119,Y -281.395,Z 94.580,A 103.992,B 90.000,C 0.000} C_DIS
LIN {X 70.014,Y -281.421,Z 97.077,A 103.971,B 90.000,C 0.000} C_DIS
LIN {X 69.962,Y -281.434,Z 98.432,A 103.960,B 90.000,C 0.000} C_DIS
LIN {X 70.012,Y -281.422,Z 98.556,A 103.970,B 90.000,C 0.000} C_DIS
LIN {X 69.899,Y -281.450,Z 101.053,A 103.947,B 90.000,C 0.000} C_DIS
LIN {X 69.793,Y -281.476,Z 103.550,A 103.926,B 90.000,C 0.000} C_DIS
LIN {X 69.681,Y -281.504,Z 105.453,A 103.903,B 90.000,C 0.000} C_DIS
LIN {X 69.607,Y -281.522,Z 105.577,A 103.888,B 90.000,C 0.000} C_DIS
LIN {X 69.326,Y -281.592,Z 105.604,A 103.831,B 90.000,C 0.000} C_DIS
LIN {X 68.280,Y -281.847,Z 105.577,A 103.618,B 90.000,C 0.000} C_DIS
LIN {X 68.105,Y -281.889,Z 105.629,A 103.583,B 90.000,C 0.000} C_DIS
LIN {X 66.200,Y -282.343,Z 105.525,A 103.196,B 90.000,C 0.000} C_DIS
LIN {X 65.923,Y -282.408,Z 105.461,A 103.139,B 90.000,C 0.000} C_DIS
LIN {X 65.915,Y -282.410,Z 104.508,A 103.138,B 90.000,C 0.000} C_DIS
LIN {X 65.893,Y -282.415,Z 104.351,A 103.133,B 90.000,C 0.000} C_DIS
LIN {X 65.873,Y -282.420,Z 104.287,A 103.129,B 90.000,C 0.000} C_DIS
LIN {X 65.974,Y -282.396,Z 101.913,A 103.150,B 90.000,C 0.000} C_DIS
LIN {X 65.924,Y -282.408,Z 101.686,A 103.140,B 90.000,C 0.000} C_DIS
LIN {X 66.032,Y -282.382,Z 99.347,A 103.162,B 90.000,C 0.000} C_DIS
LIN {X 66.013,Y -282.387,Z 99.288,A 103.158,B 90.000,C 0.000} C_DIS
LIN {X 65.985,Y -282.393,Z 99.160,A 103.152,B 90.000,C 0.000} C_DIS
LIN {X 66.072,Y -282.373,Z 96.661,A 103.170,B 90.000,C 0.000} C_DIS
LIN {X 66.137,Y -282.358,Z 94.162,A 103.183,B 90.000,C 0.000} C_DIS
LIN {X 66.232,Y -282.335,Z 91.664,A 103.202,B 90.000,C 0.000} C_DIS
LIN {X 66.252,Y -282.331,Z 91.385,A 103.206,B 90.000,C 0.000} C_DIS
LIN {X 66.225,Y -282.337,Z 91.322,A 103.201,B 90.000,C 0.000} C_DIS
LIN {X 66.200,Y -282.343,Z 91.166,A 103.196,B 90.000,C 0.000} C_DIS
LIN {X 66.304,Y -282.319,Z 88.727,A 103.217,B 90.000,C 0.000} C_DIS
LIN {X 65.847,Y -280.372,Z 88.727,A 103.217,B 90.000,C 0.000} C_DIS
WAIT SEC 0.1
RET=EKI_SetBool("oxy","torchState",FALSE)
RET = EKI_Send("oxy","torchState")
LIN {X 61.732,Y -262.848,Z 88.727,A 103.217,B 90.000,C 0.000} C_DIS
LIN {X 67.864,Y -261.332,Z 91.018,A 104.557,B 90.000,C 0.000} C_DIS
LIN {X 72.389,Y -278.754,Z 91.018,A 104.557,B 90.000,C 0.000} C_DIS
LIN {X 72.891,Y -280.690,Z 91.018,A 104.557,B 90.000,C 0.000} C_DIS
WAIT SEC 1
RET=EKI_SetBool("oxy","torchState",TRUE)
RET = EKI_Send("oxy","torchState")
LIN {X 72.975,Y -280.668,Z 88.519,A 104.574,B 90.000,C 0.000} C_DIS
LIN {X 73.043,Y -280.650,Z 87.183,A 104.588,B 90.000,C 0.000} C_DIS
LIN {X 72.998,Y -280.662,Z 86.991,A 104.579,B 90.000,C 0.000} C_DIS
LIN {X 73.072,Y -280.643,Z 85.456,A 104.594,B 90.000,C 0.000} C_DIS
LIN {X 73.072,Y -280.643,Z 85.456,A 104.594,B 90.000,C 0.000} C_DIS
LIN {X 75.488,Y -280.001,Z 85.416,A 105.088,B 90.000,C 0.000} C_DIS
LIN {X 77.166,Y -279.545,Z 85.490,A 105.432,B 90.000,C 0.000} C_DIS
LIN {X 77.165,Y -279.545,Z 87.861,A 105.431,B 90.000,C 0.000} C_DIS
LIN {X 77.063,Y -279.574,Z 90.234,A 105.411,B 90.000,C 0.000} C_DIS
LIN {X 77.087,Y -279.567,Z 90.355,A 105.416,B 90.000,C 0.000} C_DIS
LIN {X 77.114,Y -279.559,Z 90.414,A 105.421,B 90.000,C 0.000} C_DIS
LIN {X 77.008,Y -279.589,Z 92.229,A 105.399,B 90.000,C 0.000} C_DIS
LIN {X 77.034,Y -279.581,Z 92.319,A 105.405,B 90.000,C 0.000} C_DIS
LIN {X 77.055,Y -279.576,Z 92.478,A 105.409,B 90.000,C 0.000} C_DIS
LIN {X 76.947,Y -279.605,Z 94.976,A 105.387,B 90.000,C 0.000} C_DIS
LIN {X 76.900,Y -279.618,Z 96.265,A 105.377,B 90.000,C 0.000} C_DIS
LIN {X 76.924,Y -279.612,Z 96.329,A 105.382,B 90.000,C 0.000} C_DIS
LIN {X 76.948,Y -279.605,Z 96.453,A 105.387,B 90.000,C 0.000} C_DIS
LIN {X 76.845,Y -279.633,Z 98.257,A 105.366,B 90.000,C 0.000} C_DIS
LIN {X 76.895,Y -279.620,Z 98.378,A 105.376,B 90.000,C 0.000} C_DIS
LIN {X 76.791,Y -279.648,Z 100.241,A 105.355,B 90.000,C 0.000} C_DIS
LIN {X 76.836,Y -279.636,Z 100.434,A 105.364,B 90.000,C 0.000} C_DIS
LIN {X 76.760,Y -279.657,Z 102.650,A 105.349,B 90.000,C 0.000} C_DIS
LIN {X 76.557,Y -279.713,Z 103.311,A 105.307,B 90.000,C 0.000} C_DIS
LIN {X 76.237,Y -279.800,Z 103.803,A 105.241,B 90.000,C 0.000} C_DIS
LIN {X 76.105,Y -279.836,Z 104.067,A 105.214,B 90.000,C 0.000} C_DIS
LIN {X 75.445,Y -280.014,Z 105.091,A 105.079,B 90.000,C 0.000} C_DIS
LIN {X 75.358,Y -280.038,Z 105.206,A 105.062,B 90.000,C 0.000} C_DIS
LIN {X 75.272,Y -280.061,Z 105.288,A 105.044,B 90.000,C 0.000} C_DIS
LIN {X 75.221,Y -280.075,Z 105.307,A 105.033,B 90.000,C 0.000} C_DIS
LIN {X 74.982,Y -280.139,Z 105.564,A 104.985,B 90.000,C 0.000} C_DIS
LIN {X 74.864,Y -280.170,Z 105.660,A 104.960,B 90.000,C 0.000} C_DIS
LIN {X 74.782,Y -280.192,Z 105.712,A 104.944,B 90.000,C 0.000} C_DIS
LIN {X 74.562,Y -280.251,Z 105.759,A 104.899,B 90.000,C 0.000} C_DIS
LIN {X 74.135,Y -280.364,Z 105.794,A 104.811,B 90.000,C 0.000} C_DIS
LIN {X 72.814,Y -280.710,Z 105.704,A 104.542,B 90.000,C 0.000} C_DIS
LIN {X 72.617,Y -280.761,Z 105.637,A 104.501,B 90.000,C 0.000} C_DIS
LIN {X 72.572,Y -280.773,Z 105.528,A 104.492,B 90.000,C 0.000} C_DIS
LIN {X 72.577,Y -280.771,Z 103.669,A 104.493,B 90.000,C 0.000} C_DIS
LIN {X 72.559,Y -280.776,Z 103.541,A 104.490,B 90.000,C 0.000} C_DIS
LIN {X 72.628,Y -280.758,Z 101.042,A 104.504,B 90.000,C 0.000} C_DIS
LIN {X 72.657,Y -280.751,Z 99.985,A 104.510,B 90.000,C 0.000} C_DIS
LIN {X 72.612,Y -280.762,Z 99.793,A 104.500,B 90.000,C 0.000} C_DIS
LIN {X 72.706,Y -280.738,Z 97.295,A 104.520,B 90.000,C 0.000} C_DIS
LIN {X 72.770,Y -280.722,Z 94.796,A 104.533,B 90.000,C 0.000} C_DIS
LIN {X 72.868,Y -280.696,Z 92.298,A 104.553,B 90.000,C 0.000} C_DIS
LIN {X 72.882,Y -280.692,Z 92.068,A 104.556,B 90.000,C 0.000} C_DIS
LIN {X 72.857,Y -280.699,Z 91.891,A 104.550,B 90.000,C 0.000} C_DIS
LIN {X 72.832,Y -280.705,Z 91.828,A 104.545,B 90.000,C 0.000} C_DIS
LIN {X 72.891,Y -280.690,Z 91.018,A 104.557,B 90.000,C 0.000} C_DIS
LIN {X 72.389,Y -278.754,Z 91.018,A 104.557,B 90.000,C 0.000} C_DIS
WAIT SEC 0.1
RET=EKI_SetBool("oxy","torchState",FALSE)
RET = EKI_Send("oxy","torchState")
LIN {X 67.864,Y -261.332,Z 91.018,A 104.557,B 90.000,C 0.000} C_DIS
LIN {X 68.033,Y -261.288,Z 85.456,A 104.594,B 90.000,C 0.000} C_DIS
LIN {X 72.568,Y -278.707,Z 85.456,A 104.594,B 90.000,C 0.000} C_DIS
LIN {X 73.072,Y -280.643,Z 85.456,A 104.594,B 90.000,C 0.000} C_DIS
WAIT SEC 1
RET=EKI_SetBool("oxy","torchState",TRUE)
RET = EKI_Send("oxy","torchState")
LIN {X 73.072,Y -280.643,Z 85.456,A 104.594,B 90.000,C 0.000} C_DIS
LIN {X 72.568,Y -278.707,Z 85.456,A 104.594,B 90.000,C 0.000} C_DIS
WAIT SEC 0.1
RET=EKI_SetBool("oxy","torchState",FALSE)
RET = EKI_Send("oxy","torchState")
LIN {X 68.033,Y -261.288,Z 85.456,A 104.594,B 90.000,C 0.000} C_DIS
LIN {X 74.423,Y -259.540,Z 85.764,A 106.000,B 90.000,C 0.000} C_DIS
LIN {X 79.385,Y -276.843,Z 85.764,A 106.000,B 90.000,C 0.000} C_DIS
LIN {X 79.936,Y -278.766,Z 85.764,A 106.000,B 90.000,C 0.000} C_DIS
WAIT SEC 1
RET=EKI_SetBool("oxy","torchState",TRUE)
RET = EKI_Send("oxy","torchState")
LIN {X 79.869,Y -278.785,Z 88.263,A 105.987,B 90.000,C 0.000} C_DIS
LIN {X 79.797,Y -278.805,Z 90.762,A 105.972,B 90.000,C 0.000} C_DIS
LIN {X 79.750,Y -278.819,Z 91.428,A 105.962,B 90.000,C 0.000} C_DIS
LIN {X 79.792,Y -278.807,Z 91.621,A 105.971,B 90.000,C 0.000} C_DIS
LIN {X 79.724,Y -278.826,Z 94.120,A 105.957,B 90.000,C 0.000} C_DIS
LIN {X 79.634,Y -278.852,Z 96.616,A 105.938,B 90.000,C 0.000} C_DIS
LIN {X 79.658,Y -278.845,Z 96.645,A 105.943,B 90.000,C 0.000} C_DIS
LIN {X 79.696,Y -278.834,Z 96.761,A 105.951,B 90.000,C 0.000} C_DIS
LIN {X 79.628,Y -278.854,Z 97.135,A 105.937,B 90.000,C 0.000} C_DIS
LIN {X 79.706,Y -278.832,Z 97.410,A 105.953,B 90.000,C 0.000} C_DIS
LIN {X 80.049,Y -278.733,Z 96.986,A 106.024,B 90.000,C 0.000} C_DIS
LIN {X 80.100,Y -278.718,Z 96.910,A 106.034,B 90.000,C 0.000} C_DIS
LIN {X 80.209,Y -278.687,Z 96.671,A 106.056,B 90.000,C 0.000} C_DIS
LIN {X 80.401,Y -278.632,Z 96.349,A 106.096,B 90.000,C 0.000} C_DIS
LIN {X 80.483,Y -278.608,Z 96.160,A 106.113,B 90.000,C 0.000} C_DIS
LIN {X 80.698,Y -278.546,Z 95.760,A 106.157,B 90.000,C 0.000} C_DIS
LIN {X 81.416,Y -278.337,Z 94.540,A 106.305,B 90.000,C 0.000} C_DIS
LIN {X 81.466,Y -278.322,Z 94.487,A 106.315,B 90.000,C 0.000} C_DIS
LIN {X 81.739,Y -278.242,Z 93.996,A 106.371,B 90.000,C 0.000} C_DIS
LIN {X 82.445,Y -278.034,Z 92.745,A 106.517,B 90.000,C 0.000} C_DIS
LIN {X 82.523,Y -278.011,Z 92.570,A 106.533,B 90.000,C 0.000} C_DIS
LIN {X 82.667,Y -277.968,Z 92.354,A 106.562,B 90.000,C 0.000} C_DIS
LIN {X 82.861,Y -277.910,Z 91.927,A 106.602,B 90.000,C 0.000} C_DIS
LIN {X 83.018,Y -277.863,Z 91.685,A 106.635,B 90.000,C 0.000} C_DIS
LIN {X 83.212,Y -277.805,Z 91.260,A 106.675,B 90.000,C 0.000} C_DIS
LIN {X 83.375,Y -277.756,Z 90.979,A 106.708,B 90.000,C 0.000} C_DIS
LIN {X 84.327,Y -277.469,Z 88.705,A 106.905,B 90.000,C 0.000} C_DIS
LIN {X 84.551,Y -277.401,Z 87.693,A 106.951,B 90.000,C 0.000} C_DIS
LIN {X 84.604,Y -277.385,Z 87.093,A 106.962,B 90.000,C 0.000} C_DIS
LIN {X 84.566,Y -277.396,Z 86.828,A 106.954,B 90.000,C 0.000} C_DIS
LIN {X 84.495,Y -277.418,Z 86.625,A 106.940,B 90.000,C 0.000} C_DIS
LIN {X 84.335,Y -277.466,Z 86.316,A 106.907,B 90.000,C 0.000} C_DIS
LIN {X 83.951,Y -277.583,Z 85.928,A 106.827,B 90.000,C 0.000} C_DIS
LIN {X 83.191,Y -277.812,Z 85.711,A 106.670,B 90.000,C 0.000} C_DIS
LIN {X 80.797,Y -278.517,Z 85.563,A 106.177,B 90.000,C 0.000} C_DIS
LIN {X 80.153,Y -278.703,Z 85.546,A 106.045,B 90.000,C 0.000} C_DIS
LIN {X 80.100,Y -278.718,Z 85.572,A 106.034,B 90.000,C 0.000} C_DIS
LIN {X 80.018,Y -278.742,Z 85.633,A 106.017,B 90.000,C 0.000} C_DIS
LIN {X 79.965,Y -278.757,Z 85.646,A 106.006,B 90.000,C 0.000} C_DIS
LIN {X 79.936,Y -278.766,Z 85.764,A 106.000,B 90.000,C 0.000} C_DIS
LIN {X 79.385,Y -276.843,Z 85.764,A 106.000,B 90.000,C 0.000} C_DIS
WAIT SEC 0.1
RET=EKI_SetBool("oxy","torchState",FALSE)
RET = EKI_Send("oxy","torchState")
LIN {X 74.423,Y -259.540,Z 85.764,A 106.000,B 90.000,C 0.000} C_DIS
LIN {X 80.085,Y -257.850,Z 87.145,A 107.254,B 90.000,C 0.000} C_DIS
LIN {X 85.424,Y -275.040,Z 87.145,A 107.254,B 90.000,C 0.000} C_DIS
LIN {X 86.017,Y -276.950,Z 87.145,A 107.254,B 90.000,C 0.000} C_DIS
WAIT SEC 1
RET=EKI_SetBool("oxy","torchState",TRUE)
RET = EKI_Send("oxy","torchState")
LIN {X 86.319,Y -276.855,Z 86.429,A 107.317,B 90.000,C 0.000} C_DIS
LIN {X 86.407,Y -276.828,Z 86.330,A 107.335,B 90.000,C 0.000} C_DIS
LIN {X 86.501,Y -276.799,Z 86.157,A 107.354,B 90.000,C 0.000} C_DIS
LIN {X 87.236,Y -276.568,Z 85.446,A 107.507,B 90.000,C 0.000} C_DIS
LIN {X 87.345,Y -276.534,Z 85.415,A 107.529,B 90.000,C 0.000} C_DIS
LIN {X 87.725,Y -276.413,Z 85.225,A 107.608,B 90.000,C 0.000} C_DIS
LIN {X 88.646,Y -276.119,Z 85.062,A 107.799,B 90.000,C 0.000} C_DIS
LIN {X 89.783,Y -275.752,Z 85.319,A 108.035,B 90.000,C 0.000} C_DIS
LIN {X 89.986,Y -275.686,Z 85.431,A 108.077,B 90.000,C 0.000} C_DIS
LIN {X 90.270,Y -275.593,Z 85.634,A 108.136,B 90.000,C 0.000} C_DIS
LIN {X 90.819,Y -275.412,Z 86.202,A 108.250,B 90.000,C 0.000} C_DIS
LIN {X 90.847,Y -275.403,Z 86.239,A 108.256,B 90.000,C 0.000} C_DIS
LIN {X 91.193,Y -275.289,Z 86.973,A 108.328,B 90.000,C 0.000} C_DIS
LIN {X 91.248,Y -275.270,Z 87.201,A 108.340,B 90.000,C 0.000} C_DIS
LIN {X 91.290,Y -275.256,Z 87.567,A 108.348,B 90.000,C 0.000} C_DIS
LIN {X 91.323,Y -275.246,Z 87.638,A 108.355,B 90.000,C 0.000} C_DIS
LIN {X 91.199,Y -275.287,Z 88.698,A 108.329,B 90.000,C 0.000} C_DIS
LIN {X 90.806,Y -275.417,Z 89.527,A 108.248,B 90.000,C 0.000} C_DIS
LIN {X 90.756,Y -275.433,Z 89.550,A 108.237,B 90.000,C 0.000} C_DIS
LIN {X 90.226,Y -275.607,Z 90.127,A 108.127,B 90.000,C 0.000} C_DIS
LIN {X 90.053,Y -275.664,Z 90.241,A 108.091,B 90.000,C 0.000} C_DIS
LIN {X 89.729,Y -275.769,Z 90.406,A 108.024,B 90.000,C 0.000} C_DIS
LIN {X 88.883,Y -276.043,Z 90.638,A 107.848,B 90.000,C 0.000} C_DIS
LIN {X 88.092,Y -276.297,Z 90.586,A 107.684,B 90.000,C 0.000} C_DIS
LIN {X 87.473,Y -276.493,Z 90.384,A 107.556,B 90.000,C 0.000} C_DIS
LIN {X 87.182,Y -276.585,Z 90.240,A 107.495,B 90.000,C 0.000} C_DIS
LIN {X 86.639,Y -276.756,Z 89.759,A 107.383,B 90.000,C 0.000} C_DIS
LIN {X 86.503,Y -276.798,Z 89.582,A 107.355,B 90.000,C 0.000} C_DIS
LIN {X 86.145,Y -276.910,Z 88.990,A 107.281,B 90.000,C 0.000} C_DIS
LIN {X 86.106,Y -276.922,Z 88.947,A 107.272,B 90.000,C 0.000} C_DIS
LIN {X 86.045,Y -276.941,Z 88.648,A 107.260,B 90.000,C 0.000} C_DIS
LIN {X 85.964,Y -276.966,Z 87.626,A 107.243,B 90.000,C 0.000} C_DIS
LIN {X 86.017,Y -276.950,Z 87.145,A 107.254,B 90.000,C 0.000} C_DIS
LIN {X 85.424,Y -275.040,Z 87.145,A 107.254,B 90.000,C 0.000} C_DIS
WAIT SEC 0.1
RET=EKI_SetBool("oxy","torchState",FALSE)
RET = EKI_Send("oxy","torchState")
LIN {X 80.085,Y -257.850,Z 87.145,A 107.254,B 90.000,C 0.000} C_DIS
LIN {X 84.430,Y -256.460,Z 91.844,A 108.222,B 90.000,C 0.000} C_DIS
LIN {X 90.059,Y -273.557,Z 91.844,A 108.222,B 90.000,C 0.000} C_DIS
LIN {X 90.684,Y -275.457,Z 91.844,A 108.222,B 90.000,C 0.000} C_DIS
WAIT SEC 1
RET=EKI_SetBool("oxy","torchState",TRUE)
RET = EKI_Send("oxy","torchState")
LIN {X 90.674,Y -275.460,Z 91.890,A 108.220,B 90.000,C 0.000} C_DIS
LIN {X 90.649,Y -275.468,Z 91.948,A 108.215,B 90.000,C 0.000} C_DIS
LIN {X 90.316,Y -275.578,Z 92.249,A 108.146,B 90.000,C 0.000} C_DIS
LIN {X 89.980,Y -275.687,Z 92.762,A 108.076,B 90.000,C 0.000} C_DIS
LIN {X 89.817,Y -275.741,Z 93.274,A 108.042,B 90.000,C 0.000} C_DIS
LIN {X 89.796,Y -275.747,Z 94.149,A 108.038,B 90.000,C 0.000} C_DIS
LIN {X 90.058,Y -275.662,Z 94.922,A 108.092,B 90.000,C 0.000} C_DIS
LIN {X 90.215,Y -275.611,Z 95.227,A 108.125,B 90.000,C 0.000} C_DIS
LIN {X 90.634,Y -275.473,Z 95.807,A 108.212,B 90.000,C 0.000} C_DIS
LIN {X 90.702,Y -275.451,Z 95.938,A 108.226,B 90.000,C 0.000} C_DIS
LIN {X 91.607,Y -275.151,Z 97.209,A 108.414,B 90.000,C 0.000} C_DIS
LIN {X 91.674,Y -275.129,Z 97.349,A 108.428,B 90.000,C 0.000} C_DIS
LIN {X 92.015,Y -275.015,Z 97.808,A 108.499,B 90.000,C 0.000} C_DIS
LIN {X 92.037,Y -275.008,Z 97.844,A 108.504,B 90.000,C 0.000} C_DIS
LIN {X 92.068,Y -274.997,Z 97.952,A 108.510,B 90.000,C 0.000} C_DIS
LIN {X 92.524,Y -274.844,Z 98.538,A 108.605,B 90.000,C 0.000} C_DIS
LIN {X 92.676,Y -274.793,Z 98.790,A 108.637,B 90.000,C 0.000} C_DIS
LIN {X 93.651,Y -274.462,Z 100.255,A 108.841,B 90.000,C 0.000} C_DIS
LIN {X 93.992,Y -274.346,Z 100.714,A 108.912,B 90.000,C 0.000} C_DIS
LIN {X 94.059,Y -274.323,Z 100.854,A 108.926,B 90.000,C 0.000} C_DIS
LIN {X 95.242,Y -273.914,Z 102.618,A 109.173,B 90.000,C 0.000} C_DIS
LIN {X 95.444,Y -273.844,Z 102.927,A 109.215,B 90.000,C 0.000} C_DIS
LIN {X 95.501,Y -273.824,Z 102.986,A 109.227,B 90.000,C 0.000} C_DIS
LIN {X 95.712,Y -273.750,Z 103.311,A 109.271,B 90.000,C 0.000} C_DIS
LIN {X 95.805,Y -273.718,Z 103.419,A 109.291,B 90.000,C 0.000} C_DIS
LIN {X 96.893,Y -273.334,Z 105.063,A 109.519,B 90.000,C 0.000} C_DIS
LIN {X 97.322,Y -273.182,Z 105.658,A 109.609,B 90.000,C 0.000} C_DIS
LIN {X 97.379,Y -273.162,Z 105.717,A 109.621,B 90.000,C 0.000} C_DIS
LIN {X 97.402,Y -273.153,Z 105.774,A 109.625,B 90.000,C 0.000} C_DIS
LIN {X 97.418,Y -273.148,Z 105.831,A 109.629,B 90.000,C 0.000} C_DIS
LIN {X 98.701,Y -272.687,Z 107.682,A 109.898,B 90.000,C 0.000} C_DIS
LIN {X 98.768,Y -272.663,Z 107.818,A 109.912,B 90.000,C 0.000} C_DIS
LIN {X 98.824,Y -272.642,Z 107.879,A 109.924,B 90.000,C 0.000} C_DIS
LIN {X 98.848,Y -272.634,Z 107.936,A 109.929,B 90.000,C 0.000} C_DIS
LIN {X 98.863,Y -272.628,Z 107.993,A 109.932,B 90.000,C 0.000} C_DIS
LIN {X 100.074,Y -272.186,Z 109.747,A 110.187,B 90.000,C 0.000} C_DIS
LIN {X 100.998,Y -271.845,Z 111.095,A 110.381,B 90.000,C 0.000} C_DIS
LIN {X 101.064,Y -271.820,Z 111.232,A 110.395,B 90.000,C 0.000} C_DIS
LIN {X 101.121,Y -271.799,Z 111.293,A 110.407,B 90.000,C 0.000} C_DIS
LIN {X 101.331,Y -271.720,Z 111.610,A 110.452,B 90.000,C 0.000} C_DIS
LIN {X 101.744,Y -271.566,Z 112.286,A 110.539,B 90.000,C 0.000} C_DIS
LIN {X 101.811,Y -271.541,Z 112.427,A 110.553,B 90.000,C 0.000} C_DIS
LIN {X 101.867,Y -271.520,Z 112.488,A 110.565,B 90.000,C 0.000} C_DIS
LIN {X 101.891,Y -271.511,Z 112.545,A 110.570,B 90.000,C 0.000} C_DIS
LIN {X 101.903,Y -271.507,Z 112.601,A 110.572,B 90.000,C 0.000} C_DIS
LIN {X 102.503,Y -271.281,Z 113.394,A 110.699,B 90.000,C 0.000} C_DIS
LIN {X 102.560,Y -271.259,Z 113.455,A 110.711,B 90.000,C 0.000} C_DIS
LIN {X 102.691,Y -271.209,Z 113.526,A 110.739,B 90.000,C 0.000} C_DIS
LIN {X 102.847,Y -271.150,Z 113.671,A 110.772,B 90.000,C 0.000} C_DIS
LIN {X 103.732,Y -270.813,Z 113.908,A 110.959,B 90.000,C 0.000} C_DIS
LIN {X 104.244,Y -270.616,Z 113.953,A 111.067,B 90.000,C 0.000} C_DIS
LIN {X 104.682,Y -270.447,Z 113.856,A 111.160,B 90.000,C 0.000} C_DIS
LIN {X 105.159,Y -270.262,Z 113.638,A 111.261,B 90.000,C 0.000} C_DIS
LIN {X 105.530,Y -270.117,Z 113.336,A 111.340,B 90.000,C 0.000} C_DIS
LIN {X 105.907,Y -269.970,Z 112.760,A 111.420,B 90.000,C 0.000} C_DIS
LIN {X 106.069,Y -269.906,Z 112.237,A 111.454,B 90.000,C 0.000} C_DIS
LIN {X 106.134,Y -269.881,Z 111.520,A 111.468,B 90.000,C 0.000} C_DIS
LIN {X 105.871,Y -269.984,Z 110.513,A 111.412,B 90.000,C 0.000} C_DIS
LIN {X 105.742,Y -270.034,Z 110.212,A 111.385,B 90.000,C 0.000} C_DIS
LIN {X 105.689,Y -270.055,Z 110.135,A 111.373,B 90.000,C 0.000} C_DIS
LIN {X 104.722,Y -270.432,Z 108.649,A 111.168,B 90.000,C 0.000} C_DIS
LIN {X 104.098,Y -270.673,Z 107.768,A 111.036,B 90.000,C 0.000} C_DIS
LIN {X 104.042,Y -270.694,Z 107.708,A 111.024,B 90.000,C 0.000} C_DIS
LIN {X 104.018,Y -270.703,Z 107.651,A 111.019,B 90.000,C 0.000} C_DIS
LIN {X 104.003,Y -270.709,Z 107.595,A 111.016,B 90.000,C 0.000} C_DIS
LIN {X 103.312,Y -270.973,Z 106.504,A 110.870,B 90.000,C 0.000} C_DIS
LIN {X 102.740,Y -271.191,Z 105.731,A 110.749,B 90.000,C 0.000} C_DIS
LIN {X 102.595,Y -271.246,Z 105.546,A 110.718,B 90.000,C 0.000} C_DIS
LIN {X 102.568,Y -271.256,Z 105.433,A 110.713,B 90.000,C 0.000} C_DIS
LIN {X 101.184,Y -271.775,Z 103.416,A 110.421,B 90.000,C 0.000} C_DIS
LIN {X 101.160,Y -271.784,Z 103.384,A 110.416,B 90.000,C 0.000} C_DIS
LIN {X 101.129,Y -271.796,Z 103.270,A 110.409,B 90.000,C 0.000} C_DIS
LIN {X 100.839,Y -271.903,Z 102.872,A 110.348,B 90.000,C 0.000} C_DIS
LIN {X 100.798,Y -271.919,Z 102.787,A 110.339,B 90.000,C 0.000} C_DIS
LIN {X 100.371,Y -272.077,Z 102.206,A 110.249,B 90.000,C 0.000} C_DIS
LIN {X 99.718,Y -272.316,Z 101.222,A 110.112,B 90.000,C 0.000} C_DIS
LIN {X 99.703,Y -272.322,Z 101.165,A 110.109,B 90.000,C 0.000} C_DIS
LIN {X 99.680,Y -272.331,Z 101.108,A 110.104,B 90.000,C 0.000} C_DIS
LIN {X 99.623,Y -272.351,Z 101.049,A 110.092,B 90.000,C 0.000} C_DIS
LIN {X 99.196,Y -272.507,Z 100.454,A 110.002,B 90.000,C 0.000} C_DIS
LIN {X 98.114,Y -272.899,Z 98.807,A 109.775,B 90.000,C 0.000} C_DIS
LIN {X 98.018,Y -272.933,Z 98.703,A 109.755,B 90.000,C 0.000} C_DIS
LIN {X 97.807,Y -273.009,Z 98.377,A 109.710,B 90.000,C 0.000} C_DIS
LIN {X 97.751,Y -273.029,Z 98.316,A 109.699,B 90.000,C 0.000} C_DIS
LIN {X 97.684,Y -273.053,Z 98.176,A 109.684,B 90.000,C 0.000} C_DIS
LIN {X 97.483,Y -273.125,Z 97.868,A 109.642,B 90.000,C 0.000} C_DIS
LIN {X 97.426,Y -273.145,Z 97.808,A 109.630,B 90.000,C 0.000} C_DIS
LIN {X 97.402,Y -273.153,Z 97.752,A 109.625,B 90.000,C 0.000} C_DIS
LIN {X 97.390,Y -273.158,Z 97.695,A 109.623,B 90.000,C 0.000} C_DIS
LIN {X 96.360,Y -273.523,Z 96.215,A 109.407,B 90.000,C 0.000} C_DIS
LIN {X 96.303,Y -273.543,Z 96.154,A 109.395,B 90.000,C 0.000} C_DIS
LIN {X 96.236,Y -273.567,Z 96.014,A 109.381,B 90.000,C 0.000} C_DIS
LIN {X 95.567,Y -273.801,Z 95.106,A 109.241,B 90.000,C 0.000} C_DIS
LIN {X 95.536,Y -273.812,Z 94.999,A 109.234,B 90.000,C 0.000} C_DIS
LIN {X 95.515,Y -273.819,Z 94.964,A 109.230,B 90.000,C 0.000} C_DIS
LIN {X 94.352,Y -274.222,Z 93.237,A 108.987,B 90.000,C 0.000} C_DIS
LIN {X 94.324,Y -274.232,Z 93.200,A 108.981,B 90.000,C 0.000} C_DIS
LIN {X 94.261,Y -274.253,Z 93.139,A 108.968,B 90.000,C 0.000} C_DIS
LIN {X 94.194,Y -274.276,Z 92.999,A 108.954,B 90.000,C 0.000} C_DIS
LIN {X 93.992,Y -274.346,Z 92.690,A 108.912,B 90.000,C 0.000} C_DIS
LIN {X 93.858,Y -274.391,Z 92.520,A 108.884,B 90.000,C 0.000} C_DIS
LIN {X 93.638,Y -274.466,Z 92.296,A 108.838,B 90.000,C 0.000} C_DIS
LIN {X 93.550,Y -274.496,Z 92.172,A 108.819,B 90.000,C 0.000} C_DIS
LIN {X 93.282,Y -274.588,Z 91.934,A 108.764,B 90.000,C 0.000} C_DIS
LIN {X 92.896,Y -274.719,Z 91.692,A 108.683,B 90.000,C 0.000} C_DIS
LIN {X 92.008,Y -275.017,Z 91.444,A 108.498,B 90.000,C 0.000} C_DIS
LIN {X 90.972,Y -275.362,Z 91.723,A 108.282,B 90.000,C 0.000} C_DIS
LIN {X 90.684,Y -275.457,Z 91.844,A 108.222,B 90.000,C 0.000} C_DIS
LIN {X 90.059,Y -273.557,Z 91.844,A 108.222,B 90.000,C 0.000} C_DIS
WAIT SEC 0.1
RET=EKI_SetBool("oxy","torchState",FALSE)
RET = EKI_Send("oxy","torchState")
LIN {X 84.430,Y -256.460,Z 91.844,A 108.222,B 90.000,C 0.000} C_DIS
LIN {X 87.218,Y -255.525,Z 90.127,A 108.846,B 90.000,C 0.000} C_DIS
LIN {X 93.033,Y -272.560,Z 90.127,A 108.846,B 90.000,C 0.000} C_DIS
LIN {X 93.679,Y -274.453,Z 90.127,A 108.846,B 90.000,C 0.000} C_DIS
WAIT SEC 1
RET=EKI_SetBool("oxy","torchState",TRUE)
RET = EKI_Send("oxy","torchState")
LIN {X 93.723,Y -274.438,Z 90.213,A 108.855,B 90.000,C 0.000} C_DIS
LIN {X 93.798,Y -274.412,Z 90.298,A 108.871,B 90.000,C 0.000} C_DIS
LIN {X 94.020,Y -274.336,Z 90.469,A 108.918,B 90.000,C 0.000} C_DIS
LIN {X 94.153,Y -274.290,Z 90.611,A 108.945,B 90.000,C 0.000} C_DIS
LIN {X 94.261,Y -274.253,Z 90.696,A 108.968,B 90.000,C 0.000} C_DIS
LIN {X 94.960,Y -274.012,Z 91.094,A 109.114,B 90.000,C 0.000} C_DIS
LIN {X 97.145,Y -273.245,Z 92.037,A 109.571,B 90.000,C 0.000} C_DIS
LIN {X 99.315,Y -272.464,Z 93.000,A 110.027,B 90.000,C 0.000} C_DIS
LIN {X 101.478,Y -271.666,Z 93.967,A 110.483,B 90.000,C 0.000} C_DIS
LIN {X 102.864,Y -271.144,Z 94.658,A 110.775,B 90.000,C 0.000} C_DIS
LIN {X 103.891,Y -270.752,Z 95.091,A 110.992,B 90.000,C 0.000} C_DIS
LIN {X 104.562,Y -270.494,Z 95.217,A 111.134,B 90.000,C 0.000} C_DIS
LIN {X 105.200,Y -270.246,Z 95.146,A 111.270,B 90.000,C 0.000} C_DIS
LIN {X 105.424,Y -270.159,Z 95.089,A 111.317,B 90.000,C 0.000} C_DIS
LIN {X 105.927,Y -269.962,Z 94.761,A 111.424,B 90.000,C 0.000} C_DIS
LIN {X 106.113,Y -269.889,Z 94.604,A 111.463,B 90.000,C 0.000} C_DIS
LIN {X 106.519,Y -269.729,Z 94.083,A 111.550,B 90.000,C 0.000} C_DIS
LIN {X 106.762,Y -269.633,Z 93.476,A 111.601,B 90.000,C 0.000} C_DIS
LIN {X 106.819,Y -269.610,Z 92.881,A 111.613,B 90.000,C 0.000} C_DIS
LIN {X 106.763,Y -269.632,Z 92.304,A 111.602,B 90.000,C 0.000} C_DIS
LIN {X 106.707,Y -269.655,Z 92.062,A 111.590,B 90.000,C 0.000} C_DIS
LIN {X 106.532,Y -269.724,Z 91.777,A 111.552,B 90.000,C 0.000} C_DIS
LIN {X 106.487,Y -269.742,Z 91.664,A 111.543,B 90.000,C 0.000} C_DIS
LIN {X 106.195,Y -269.857,Z 91.303,A 111.481,B 90.000,C 0.000} C_DIS
LIN {X 105.689,Y -270.055,Z 90.872,A 111.373,B 90.000,C 0.000} C_DIS
LIN {X 104.971,Y -270.335,Z 90.445,A 111.221,B 90.000,C 0.000} C_DIS
LIN {X 102.806,Y -271.166,Z 89.511,A 110.763,B 90.000,C 0.000} C_DIS
LIN {X 100.650,Y -271.973,Z 88.537,A 110.308,B 90.000,C 0.000} C_DIS
LIN {X 98.489,Y -272.763,Z 87.559,A 109.854,B 90.000,C 0.000} C_DIS
LIN {X 96.569,Y -273.449,Z 86.652,A 109.451,B 90.000,C 0.000} C_DIS
LIN {X 96.040,Y -273.635,Z 86.494,A 109.340,B 90.000,C 0.000} C_DIS
LIN {X 95.519,Y -273.818,Z 86.439,A 109.231,B 90.000,C 0.000} C_DIS
LIN {X 94.965,Y -274.010,Z 86.491,A 109.115,B 90.000,C 0.000} C_DIS
LIN {X 94.638,Y -274.124,Z 86.607,A 109.047,B 90.000,C 0.000} C_DIS
LIN {X 94.194,Y -274.276,Z 86.884,A 108.954,B 90.000,C 0.000} C_DIS
LIN {X 93.669,Y -274.456,Z 87.459,A 108.844,B 90.000,C 0.000} C_DIS
LIN {X 93.615,Y -274.474,Z 87.482,A 108.833,B 90.000,C 0.000} C_DIS
LIN {X 93.561,Y -274.493,Z 87.560,A 108.822,B 90.000,C 0.000} C_DIS
LIN {X 93.317,Y -274.576,Z 88.268,A 108.771,B 90.000,C 0.000} C_DIS
LIN {X 93.272,Y -274.591,Z 88.945,A 108.761,B 90.000,C 0.000} C_DIS
LIN {X 93.311,Y -274.578,Z 89.374,A 108.770,B 90.000,C 0.000} C_DIS
LIN {X 93.359,Y -274.562,Z 89.502,A 108.780,B 90.000,C 0.000} C_DIS
LIN {X 93.679,Y -274.453,Z 90.127,A 108.846,B 90.000,C 0.000} C_DIS
LIN {X 93.033,Y -272.560,Z 90.127,A 108.846,B 90.000,C 0.000} C_DIS
WAIT SEC 0.1
RET=EKI_SetBool("oxy","torchState",FALSE)
RET = EKI_Send("oxy","torchState")
LIN {X 87.218,Y -255.525,Z 90.127,A 108.846,B 90.000,C 0.000} C_DIS
LIN {X 82.595,Y -257.056,Z 97.811,A 107.813,B 90.000,C 0.000} C_DIS
LIN {X 88.102,Y -274.194,Z 97.811,A 107.813,B 90.000,C 0.000} C_DIS
LIN {X 88.714,Y -276.098,Z 97.811,A 107.813,B 90.000,C 0.000} C_DIS
WAIT SEC 1
RET=EKI_SetBool("oxy","torchState",TRUE)
RET = EKI_Send("oxy","torchState")
LIN {X 88.917,Y -276.032,Z 97.925,A 107.855,B 90.000,C 0.000} C_DIS
LIN {X 89.336,Y -275.897,Z 98.321,A 107.942,B 90.000,C 0.000} C_DIS
LIN {X 89.666,Y -275.790,Z 98.833,A 108.011,B 90.000,C 0.000} C_DIS
LIN {X 89.769,Y -275.756,Z 98.961,A 108.032,B 90.000,C 0.000} C_DIS
LIN {X 90.432,Y -275.540,Z 99.897,A 108.170,B 90.000,C 0.000} C_DIS
LIN {X 90.486,Y -275.522,Z 100.053,A 108.181,B 90.000,C 0.000} C_DIS
LIN {X 90.594,Y -275.486,Z 100.218,A 108.203,B 90.000,C 0.000} C_DIS
LIN {X 90.810,Y -275.415,Z 100.633,A 108.248,B 90.000,C 0.000} C_DIS
LIN {X 90.864,Y -275.397,Z 100.710,A 108.260,B 90.000,C 0.000} C_DIS
LIN {X 90.907,Y -275.383,Z 100.753,A 108.269,B 90.000,C 0.000} C_DIS
LIN {X 91.081,Y -275.326,Z 101.222,A 108.305,B 90.000,C 0.000} C_DIS
LIN {X 91.131,Y -275.309,Z 101.450,A 108.315,B 90.000,C 0.000} C_DIS
LIN {X 91.305,Y -275.252,Z 101.848,A 108.351,B 90.000,C 0.000} C_DIS
LIN {X 91.353,Y -275.236,Z 102.076,A 108.361,B 90.000,C 0.000} C_DIS
LIN {X 91.525,Y -275.179,Z 102.474,A 108.397,B 90.000,C 0.000} C_DIS
LIN {X 91.569,Y -275.164,Z 102.701,A 108.406,B 90.000,C 0.000} C_DIS
LIN {X 91.729,Y -275.110,Z 103.100,A 108.440,B 90.000,C 0.000} C_DIS
LIN {X 91.767,Y -275.098,Z 103.327,A 108.448,B 90.000,C 0.000} C_DIS
LIN {X 92.005,Y -275.018,Z 103.953,A 108.497,B 90.000,C 0.000} C_DIS
LIN {X 92.038,Y -275.007,Z 104.196,A 108.504,B 90.000,C 0.000} C_DIS
LIN {X 92.338,Y -274.907,Z 105.091,A 108.567,B 90.000,C 0.000} C_DIS
LIN {X 92.375,Y -274.894,Z 105.319,A 108.574,B 90.000,C 0.000} C_DIS
LIN {X 92.596,Y -274.820,Z 106.058,A 108.620,B 90.000,C 0.000} C_DIS
LIN {X 92.628,Y -274.809,Z 106.277,A 108.627,B 90.000,C 0.000} C_DIS
LIN {X 93.018,Y -274.677,Z 107.677,A 108.708,B 90.000,C 0.000} C_DIS
LIN {X 93.299,Y -274.582,Z 108.676,A 108.767,B 90.000,C 0.000} C_DIS
LIN {X 93.307,Y -274.579,Z 108.789,A 108.769,B 90.000,C 0.000} C_DIS
LIN {X 93.384,Y -274.553,Z 109.017,A 108.785,B 90.000,C 0.000} C_DIS
LIN {X 93.393,Y -274.550,Z 109.131,A 108.787,B 90.000,C 0.000} C_DIS
LIN {X 93.674,Y -274.454,Z 110.130,A 108.845,B 90.000,C 0.000} C_DIS
LIN {X 93.704,Y -274.444,Z 110.374,A 108.852,B 90.000,C 0.000} C_DIS
LIN {X 94.055,Y -274.324,Z 111.492,A 108.925,B 90.000,C 0.000} C_DIS
LIN {X 94.323,Y -274.232,Z 112.488,A 108.981,B 90.000,C 0.000} C_DIS
LIN {X 94.330,Y -274.229,Z 112.601,A 108.982,B 90.000,C 0.000} C_DIS
LIN {X 94.366,Y -274.217,Z 112.715,A 108.990,B 90.000,C 0.000} C_DIS
LIN {X 94.418,Y -274.199,Z 112.815,A 109.001,B 90.000,C 0.000} C_DIS
LIN {X 94.652,Y -274.119,Z 114.198,A 109.050,B 90.000,C 0.000} C_DIS
LIN {X 94.653,Y -274.118,Z 114.422,A 109.050,B 90.000,C 0.000} C_DIS
LIN {X 94.498,Y -274.172,Z 114.653,A 109.017,B 90.000,C 0.000} C_DIS
LIN {X 94.369,Y -274.216,Z 114.776,A 108.990,B 90.000,C 0.000} C_DIS
LIN {X 94.315,Y -274.235,Z 114.792,A 108.979,B 90.000,C 0.000} C_DIS
LIN {X 94.261,Y -274.253,Z 114.817,A 108.968,B 90.000,C 0.000} C_DIS
LIN {X 94.100,Y -274.309,Z 114.937,A 108.934,B 90.000,C 0.000} C_DIS
LIN {X 93.992,Y -274.346,Z 114.981,A 108.912,B 90.000,C 0.000} C_DIS
LIN {X 93.615,Y -274.474,Z 115.171,A 108.833,B 90.000,C 0.000} C_DIS
LIN {X 93.507,Y -274.511,Z 115.202,A 108.811,B 90.000,C 0.000} C_DIS
LIN {X 93.400,Y -274.548,Z 115.217,A 108.788,B 90.000,C 0.000} C_DIS
LIN {X 92.643,Y -274.804,Z 115.473,A 108.630,B 90.000,C 0.000} C_DIS
LIN {X 92.275,Y -274.928,Z 115.507,A 108.554,B 90.000,C 0.000} C_DIS
LIN {X 92.181,Y -274.959,Z 115.550,A 108.534,B 90.000,C 0.000} C_DIS
LIN {X 91.566,Y -275.165,Z 115.714,A 108.406,B 90.000,C 0.000} C_DIS
LIN {X 91.188,Y -275.290,Z 115.793,A 108.327,B 90.000,C 0.000} C_DIS
LIN {X 91.094,Y -275.322,Z 115.844,A 108.307,B 90.000,C 0.000} C_DIS
LIN {X 89.685,Y -275.783,Z 116.191,A 108.015,B 90.000,C 0.000} C_DIS
LIN {X 89.564,Y -275.823,Z 116.202,A 107.989,B 90.000,C 0.000} C_DIS
LIN {X 89.458,Y -275.857,Z 116.240,A 107.967,B 90.000,C 0.000} C_DIS
LIN {X 89.363,Y -275.888,Z 116.294,A 107.948,B 90.000,C 0.000} C_DIS
LIN {X 87.029,Y -276.633,Z 116.789,A 107.464,B 90.000,C 0.000} C_DIS
LIN {X 85.392,Y -277.143,Z 117.070,A 107.125,B 90.000,C 0.000} C_DIS
LIN {X 85.306,Y -277.169,Z 117.099,A 107.107,B 90.000,C 0.000} C_DIS
LIN {X 82.920,Y -277.891,Z 117.286,A 106.615,B 90.000,C 0.000} C_DIS
LIN {X 80.524,Y -278.596,Z 117.380,A 106.121,B 90.000,C 0.000} C_DIS
LIN {X 78.117,Y -279.272,Z 117.363,A 105.627,B 90.000,C 0.000} C_DIS
LIN {X 75.709,Y -279.943,Z 117.331,A 105.133,B 90.000,C 0.000} C_DIS
LIN {X 73.299,Y -280.584,Z 117.161,A 104.641,B 90.000,C 0.000} C_DIS
LIN {X 73.129,Y -280.628,Z 117.148,A 104.606,B 90.000,C 0.000} C_DIS
LIN {X 72.845,Y -280.702,Z 117.064,A 104.548,B 90.000,C 0.000} C_DIS
LIN {X 72.690,Y -280.742,Z 116.698,A 104.516,B 90.000,C 0.000} C_DIS
LIN {X 72.656,Y -280.751,Z 116.470,A 104.509,B 90.000,C 0.000} C_DIS
LIN {X 72.531,Y -280.783,Z 113.974,A 104.484,B 90.000,C 0.000} C_DIS
LIN {X 72.517,Y -280.787,Z 113.626,A 104.481,B 90.000,C 0.000} C_DIS
LIN {X 72.500,Y -280.791,Z 113.526,A 104.478,B 90.000,C 0.000} C_DIS
LIN {X 72.688,Y -280.743,Z 112.646,A 104.516,B 90.000,C 0.000} C_DIS
LIN {X 72.950,Y -280.675,Z 112.332,A 104.569,B 90.000,C 0.000} C_DIS
LIN {X 73.290,Y -280.586,Z 112.032,A 104.639,B 90.000,C 0.000} C_DIS
LIN {X 74.232,Y -280.338,Z 111.394,A 104.831,B 90.000,C 0.000} C_DIS
LIN {X 74.314,Y -280.317,Z 111.350,A 104.848,B 90.000,C 0.000} C_DIS
LIN {X 74.397,Y -280.295,Z 111.289,A 104.865,B 90.000,C 0.000} C_DIS
LIN {X 74.452,Y -280.280,Z 111.264,A 104.876,B 90.000,C 0.000} C_DIS
LIN {X 74.507,Y -280.265,Z 111.248,A 104.887,B 90.000,C 0.000} C_DIS
LIN {X 74.892,Y -280.163,Z 110.938,A 104.966,B 90.000,C 0.000} C_DIS
LIN {X 76.045,Y -279.852,Z 110.291,A 105.202,B 90.000,C 0.000} C_DIS
LIN {X 76.430,Y -279.747,Z 109.972,A 105.281,B 90.000,C 0.000} C_DIS
LIN {X 76.484,Y -279.732,Z 109.956,A 105.292,B 90.000,C 0.000} C_DIS
LIN {X 76.539,Y -279.717,Z 109.931,A 105.303,B 90.000,C 0.000} C_DIS
LIN {X 76.704,Y -279.672,Z 109.810,A 105.337,B 90.000,C 0.000} C_DIS
LIN {X 76.759,Y -279.657,Z 109.785,A 105.348,B 90.000,C 0.000} C_DIS
LIN {X 76.814,Y -279.642,Z 109.769,A 105.360,B 90.000,C 0.000} C_DIS
LIN {X 77.198,Y -279.536,Z 109.459,A 105.438,B 90.000,C 0.000} C_DIS
LIN {X 77.427,Y -279.473,Z 109.341,A 105.485,B 90.000,C 0.000} C_DIS
LIN {X 77.856,Y -279.354,Z 109.001,A 105.573,B 90.000,C 0.000} C_DIS
LIN {X 77.910,Y -279.338,Z 108.989,A 105.584,B 90.000,C 0.000} C_DIS
LIN {X 77.965,Y -279.323,Z 108.963,A 105.596,B 90.000,C 0.000} C_DIS
LIN {X 78.047,Y -279.300,Z 108.903,A 105.612,B 90.000,C 0.000} C_DIS
LIN {X 78.130,Y -279.277,Z 108.859,A 105.629,B 90.000,C 0.000} C_DIS
LIN {X 78.623,Y -279.139,Z 108.492,A 105.730,B 90.000,C 0.000} C_DIS
LIN {X 78.705,Y -279.116,Z 108.448,A 105.747,B 90.000,C 0.000} C_DIS
LIN {X 78.822,Y -279.082,Z 108.352,A 105.771,B 90.000,C 0.000} C_DIS
LIN {X 79.663,Y -278.844,Z 107.753,A 105.944,B 90.000,C 0.000} C_DIS
LIN {X 79.717,Y -278.828,Z 107.737,A 105.955,B 90.000,C 0.000} C_DIS
LIN {X 79.772,Y -278.813,Z 107.712,A 105.967,B 90.000,C 0.000} C_DIS
LIN {X 80.135,Y -278.708,Z 107.441,A 106.041,B 90.000,C 0.000} C_DIS
LIN {X 80.278,Y -278.667,Z 107.291,A 106.071,B 90.000,C 0.000} C_DIS
LIN {X 80.319,Y -278.656,Z 107.257,A 106.079,B 90.000,C 0.000} C_DIS
LIN {X 80.376,Y -278.639,Z 107.196,A 106.091,B 90.000,C 0.000} C_DIS
LIN {X 80.672,Y -278.553,Z 106.983,A 106.152,B 90.000,C 0.000} C_DIS
LIN {X 80.807,Y -278.514,Z 106.912,A 106.179,B 90.000,C 0.000} C_DIS
LIN {X 80.865,Y -278.497,Z 106.852,A 106.191,B 90.000,C 0.000} C_DIS
LIN {X 80.920,Y -278.482,Z 106.826,A 106.203,B 90.000,C 0.000} C_DIS
LIN {X 80.975,Y -278.466,Z 106.810,A 106.214,B 90.000,C 0.000} C_DIS
LIN {X 81.470,Y -278.321,Z 106.427,A 106.316,B 90.000,C 0.000} C_DIS
LIN {X 83.165,Y -277.819,Z 104.659,A 106.665,B 90.000,C 0.000} C_DIS
LIN {X 83.247,Y -277.795,Z 104.567,A 106.682,B 90.000,C 0.000} C_DIS
LIN {X 83.430,Y -277.740,Z 104.420,A 106.720,B 90.000,C 0.000} C_DIS
LIN {X 84.029,Y -277.559,Z 103.620,A 106.843,B 90.000,C 0.000} C_DIS
LIN {X 84.301,Y -277.477,Z 103.331,A 106.900,B 90.000,C 0.000} C_DIS
LIN {X 84.383,Y -277.452,Z 103.270,A 106.916,B 90.000,C 0.000} C_DIS
LIN {X 84.465,Y -277.427,Z 103.185,A 106.933,B 90.000,C 0.000} C_DIS
LIN {X 84.521,Y -277.410,Z 103.100,A 106.945,B 90.000,C 0.000} C_DIS
LIN {X 84.613,Y -277.382,Z 103.000,A 106.964,B 90.000,C 0.000} C_DIS
LIN {X 85.363,Y -277.152,Z 101.961,A 107.119,B 90.000,C 0.000} C_DIS
LIN {X 85.498,Y -277.110,Z 101.821,A 107.147,B 90.000,C 0.000} C_DIS
LIN {X 85.824,Y -277.009,Z 101.306,A 107.214,B 90.000,C 0.000} C_DIS
LIN {X 85.963,Y -276.966,Z 101.156,A 107.243,B 90.000,C 0.000} C_DIS
LIN {X 86.422,Y -276.823,Z 100.487,A 107.338,B 90.000,C 0.000} C_DIS
LIN {X 86.476,Y -276.807,Z 100.454,A 107.349,B 90.000,C 0.000} C_DIS
LIN {X 86.531,Y -276.790,Z 100.431,A 107.360,B 90.000,C 0.000} C_DIS
LIN {X 86.856,Y -276.687,Z 99.940,A 107.428,B 90.000,C 0.000} C_DIS
LIN {X 86.938,Y -276.662,Z 99.857,A 107.445,B 90.000,C 0.000} C_DIS
LIN {X 87.019,Y -276.636,Z 99.797,A 107.462,B 90.000,C 0.000} C_DIS
LIN {X 87.074,Y -276.619,Z 99.669,A 107.473,B 90.000,C 0.000} C_DIS
LIN {X 87.426,Y -276.508,Z 99.137,A 107.546,B 90.000,C 0.000} C_DIS
LIN {X 87.914,Y -276.353,Z 98.227,A 107.647,B 90.000,C 0.000} C_DIS
LIN {X 88.267,Y -276.241,Z 97.862,A 107.720,B 90.000,C 0.000} C_DIS
LIN {X 88.375,Y -276.206,Z 97.812,A 107.743,B 90.000,C 0.000} C_DIS
LIN {X 88.375,Y -276.206,Z 97.812,A 107.743,B 90.000,C 0.000} C_DIS
LIN {X 88.448,Y -276.183,Z 97.755,A 107.758,B 90.000,C 0.000} C_DIS
LIN {X 88.714,Y -276.098,Z 97.811,A 107.813,B 90.000,C 0.000} C_DIS
LIN {X 88.102,Y -274.194,Z 97.811,A 107.813,B 90.000,C 0.000} C_DIS
WAIT SEC 0.1
RET=EKI_SetBool("oxy","torchState",FALSE)
RET = EKI_Send("oxy","torchState")
LIN {X 82.595,Y -257.056,Z 97.811,A 107.813,B 90.000,C 0.000} C_DIS
LIN {X 82.280,Y -257.157,Z 97.812,A 107.743,B 90.000,C 0.000} C_DIS
LIN {X 87.765,Y -274.301,Z 97.812,A 107.743,B 90.000,C 0.000} C_DIS
LIN {X 88.375,Y -276.206,Z 97.812,A 107.743,B 90.000,C 0.000} C_DIS
WAIT SEC 1
RET=EKI_SetBool("oxy","torchState",TRUE)
RET = EKI_Send("oxy","torchState")
LIN {X 88.375,Y -276.206,Z 97.812,A 107.743,B 90.000,C 0.000} C_DIS
LIN {X 87.766,Y -274.301,Z 97.812,A 107.743,B 90.000,C 0.000} C_DIS
WAIT SEC 0.1
RET=EKI_SetBool("oxy","torchState",FALSE)
RET = EKI_Send("oxy","torchState")
LIN {X 82.280,Y -257.157,Z 97.812,A 107.743,B 90.000,C 0.000} C_DIS
LIN {X 66.218,Y -261.754,Z 108.344,A 104.197,B 90.000,C 0.000} C_DIS
LIN {X 70.633,Y -279.204,Z 108.344,A 104.197,B 90.000,C 0.000} C_DIS
LIN {X 71.123,Y -281.143,Z 108.344,A 104.197,B 90.000,C 0.000} C_DIS
WAIT SEC 1
RET=EKI_SetBool("oxy","torchState",TRUE)
RET = EKI_Send("oxy","torchState")
LIN {X 68.701,Y -281.745,Z 108.199,A 103.704,B 90.000,C 0.000} C_DIS
LIN {X 66.288,Y -282.322,Z 108.081,A 103.213,B 90.000,C 0.000} C_DIS
LIN {X 66.168,Y -282.350,Z 108.132,A 103.189,B 90.000,C 0.000} C_DIS
LIN {X 64.408,Y -282.757,Z 108.024,A 102.832,B 90.000,C 0.000} C_DIS
LIN {X 62.247,Y -283.241,Z 108.021,A 102.395,B 90.000,C 0.000} C_DIS
LIN {X 59.804,Y -283.766,Z 107.926,A 101.901,B 90.000,C 0.000} C_DIS
LIN {X 59.400,Y -283.851,Z 107.910,A 101.819,B 90.000,C 0.000} C_DIS
LIN {X 59.215,Y -283.890,Z 107.959,A 101.782,B 90.000,C 0.000} C_DIS
LIN {X 57.528,Y -284.237,Z 107.960,A 101.442,B 90.000,C 0.000} C_DIS
LIN {X 57.441,Y -284.254,Z 110.382,A 101.424,B 90.000,C 0.000} C_DIS
LIN {X 57.687,Y -284.205,Z 112.870,A 101.474,B 90.000,C 0.000} C_DIS
LIN {X 58.233,Y -284.093,Z 115.081,A 101.584,B 90.000,C 0.000} C_DIS
LIN {X 58.251,Y -284.089,Z 115.166,A 101.588,B 90.000,C 0.000} C_DIS
LIN {X 58.616,Y -284.014,Z 115.958,A 101.661,B 90.000,C 0.000} C_DIS
LIN {X 58.671,Y -284.003,Z 116.035,A 101.672,B 90.000,C 0.000} C_DIS
LIN {X 58.964,Y -283.942,Z 116.558,A 101.731,B 90.000,C 0.000} C_DIS
LIN {X 59.173,Y -283.899,Z 116.866,A 101.774,B 90.000,C 0.000} C_DIS
LIN {X 59.232,Y -283.887,Z 116.925,A 101.785,B 90.000,C 0.000} C_DIS
LIN {X 59.266,Y -283.880,Z 116.968,A 101.792,B 90.000,C 0.000} C_DIS
LIN {X 59.318,Y -283.869,Z 117.084,A 101.803,B 90.000,C 0.000} C_DIS
LIN {X 59.474,Y -283.836,Z 117.165,A 101.834,B 90.000,C 0.000} C_DIS
LIN {X 59.530,Y -283.824,Z 117.261,A 101.846,B 90.000,C 0.000} C_DIS
LIN {X 59.897,Y -283.747,Z 117.718,A 101.920,B 90.000,C 0.000} C_DIS
LIN {X 59.960,Y -283.734,Z 117.779,A 101.932,B 90.000,C 0.000} C_DIS
LIN {X 61.264,Y -283.455,Z 118.795,A 102.196,B 90.000,C 0.000} C_DIS
LIN {X 61.445,Y -283.416,Z 118.885,A 102.232,B 90.000,C 0.000} C_DIS
LIN {X 61.566,Y -283.390,Z 118.973,A 102.257,B 90.000,C 0.000} C_DIS
LIN {X 63.011,Y -283.072,Z 119.723,A 102.549,B 90.000,C 0.000} C_DIS
LIN {X 63.802,Y -282.895,Z 120.078,A 102.709,B 90.000,C 0.000} C_DIS
LIN {X 64.420,Y -282.754,Z 120.021,A 102.835,B 90.000,C 0.000} C_DIS
LIN {X 66.394,Y -282.298,Z 119.250,A 103.235,B 90.000,C 0.000} C_DIS
LIN {X 66.504,Y -282.271,Z 119.205,A 103.257,B 90.000,C 0.000} C_DIS
LIN {X 66.584,Y -282.253,Z 119.144,A 103.273,B 90.000,C 0.000} C_DIS
LIN {X 66.837,Y -282.193,Z 119.002,A 103.325,B 90.000,C 0.000} C_DIS
LIN {X 67.058,Y -282.140,Z 118.910,A 103.370,B 90.000,C 0.000} C_DIS
LIN {X 67.280,Y -282.088,Z 118.732,A 103.415,B 90.000,C 0.000} C_DIS
LIN {X 67.335,Y -282.074,Z 118.718,A 103.426,B 90.000,C 0.000} C_DIS
LIN {X 67.390,Y -282.061,Z 118.693,A 103.437,B 90.000,C 0.000} C_DIS
LIN {X 67.448,Y -282.047,Z 118.632,A 103.449,B 90.000,C 0.000} C_DIS
LIN {X 68.163,Y -281.876,Z 118.066,A 103.594,B 90.000,C 0.000} C_DIS
LIN {X 68.331,Y -281.835,Z 117.957,A 103.628,B 90.000,C 0.000} C_DIS
LIN {X 68.939,Y -281.687,Z 117.180,A 103.752,B 90.000,C 0.000} C_DIS
LIN {X 69.022,Y -281.667,Z 117.096,A 103.769,B 90.000,C 0.000} C_DIS
LIN {X 69.104,Y -281.646,Z 117.035,A 103.786,B 90.000,C 0.000} C_DIS
LIN {X 69.767,Y -281.483,Z 115.907,A 103.921,B 90.000,C 0.000} C_DIS
LIN {X 70.039,Y -281.415,Z 115.332,A 103.976,B 90.000,C 0.000} C_DIS
LIN {X 70.595,Y -281.276,Z 113.682,A 104.089,B 90.000,C 0.000} C_DIS
LIN {X 70.947,Y -281.188,Z 111.892,A 104.161,B 90.000,C 0.000} C_DIS
LIN {X 71.083,Y -281.153,Z 110.638,A 104.189,B 90.000,C 0.000} C_DIS
LIN {X 71.123,Y -281.143,Z 108.344,A 104.197,B 90.000,C 0.000} C_DIS
LIN {X 70.633,Y -279.204,Z 108.344,A 104.197,B 90.000,C 0.000} C_DIS
WAIT SEC 0.1
RET=EKI_SetBool("oxy","torchState",FALSE)
RET = EKI_Send("oxy","torchState")
LIN {X 66.218,Y -261.754,Z 108.344,A 104.197,B 90.000,C 0.000} C_DIS
LIN {X 69.663,Y -260.858,Z 123.189,A 104.952,B 90.000,C 0.000} C_DIS
LIN {X 74.307,Y -278.249,Z 123.189,A 104.952,B 90.000,C 0.000} C_DIS
LIN {X 74.823,Y -280.181,Z 123.189,A 104.952,B 90.000,C 0.000} C_DIS
WAIT SEC 1
RET=EKI_SetBool("oxy","torchState",TRUE)
RET = EKI_Send("oxy","torchState")
LIN {X 75.647,Y -279.960,Z 123.018,A 105.121,B 90.000,C 0.000} C_DIS
LIN {X 76.016,Y -279.860,Z 122.976,A 105.196,B 90.000,C 0.000} C_DIS
LIN {X 77.384,Y -279.485,Z 122.706,A 105.476,B 90.000,C 0.000} C_DIS
LIN {X 78.568,Y -279.154,Z 122.542,A 105.719,B 90.000,C 0.000} C_DIS
LIN {X 80.401,Y -278.632,Z 122.561,A 106.096,B 90.000,C 0.000} C_DIS
LIN {X 82.769,Y -277.934,Z 122.955,A 106.584,B 90.000,C 0.000} C_DIS
LIN {X 85.109,Y -277.229,Z 123.480,A 107.066,B 90.000,C 0.000} C_DIS
LIN {X 87.411,Y -276.513,Z 124.142,A 107.543,B 90.000,C 0.000} C_DIS
LIN {X 89.609,Y -275.808,Z 125.101,A 107.999,B 90.000,C 0.000} C_DIS
LIN {X 90.691,Y -275.455,Z 125.744,A 108.224,B 90.000,C 0.000} C_DIS
LIN {X 91.307,Y -275.251,Z 126.118,A 108.352,B 90.000,C 0.000} C_DIS
LIN {X 91.654,Y -275.135,Z 126.313,A 108.424,B 90.000,C 0.000} C_DIS
LIN {X 91.704,Y -275.119,Z 126.365,A 108.434,B 90.000,C 0.000} C_DIS
LIN {X 92.079,Y -274.993,Z 126.631,A 108.513,B 90.000,C 0.000} C_DIS
LIN {X 92.524,Y -274.844,Z 126.935,A 108.605,B 90.000,C 0.000} C_DIS
LIN {X 92.645,Y -274.803,Z 127.051,A 108.631,B 90.000,C 0.000} C_DIS
LIN {X 92.934,Y -274.706,Z 127.281,A 108.691,B 90.000,C 0.000} C_DIS
LIN {X 93.995,Y -274.344,Z 128.077,A 108.912,B 90.000,C 0.000} C_DIS
LIN {X 95.183,Y -273.935,Z 129.158,A 109.161,B 90.000,C 0.000} C_DIS
LIN {X 95.217,Y -273.923,Z 129.272,A 109.168,B 90.000,C 0.000} C_DIS
LIN {X 95.551,Y -273.806,Z 129.618,A 109.238,B 90.000,C 0.000} C_DIS
LIN {X 96.088,Y -273.618,Z 130.324,A 109.350,B 90.000,C 0.000} C_DIS
LIN {X 96.169,Y -273.590,Z 130.410,A 109.367,B 90.000,C 0.000} C_DIS
LIN {X 96.249,Y -273.562,Z 130.452,A 109.384,B 90.000,C 0.000} C_DIS
LIN {X 96.558,Y -273.453,Z 130.979,A 109.448,B 90.000,C 0.000} C_DIS
LIN {X 96.713,Y -273.398,Z 131.211,A 109.481,B 90.000,C 0.000} C_DIS
LIN {X 97.000,Y -273.297,Z 132.230,A 109.541,B 90.000,C 0.000} C_DIS
LIN {X 97.028,Y -273.287,Z 132.767,A 109.547,B 90.000,C 0.000} C_DIS
LIN {X 96.699,Y -273.403,Z 135.223,A 109.478,B 90.000,C 0.000} C_DIS
LIN {X 95.946,Y -273.668,Z 137.592,A 109.320,B 90.000,C 0.000} C_DIS
LIN {X 95.417,Y -273.853,Z 138.794,A 109.210,B 90.000,C 0.000} C_DIS
LIN {X 95.121,Y -273.956,Z 139.322,A 109.148,B 90.000,C 0.000} C_DIS
LIN {X 94.530,Y -274.161,Z 140.252,A 109.024,B 90.000,C 0.000} C_DIS
LIN {X 94.368,Y -274.217,Z 140.444,A 108.990,B 90.000,C 0.000} C_DIS
LIN {X 94.046,Y -274.327,Z 140.946,A 108.923,B 90.000,C 0.000} C_DIS
LIN {X 93.992,Y -274.346,Z 140.964,A 108.912,B 90.000,C 0.000} C_DIS
LIN {X 93.938,Y -274.364,Z 140.998,A 108.900,B 90.000,C 0.000} C_DIS
LIN {X 92.294,Y -274.921,Z 142.796,A 108.557,B 90.000,C 0.000} C_DIS
LIN {X 92.223,Y -274.945,Z 142.870,A 108.543,B 90.000,C 0.000} C_DIS
LIN {X 91.798,Y -275.088,Z 143.210,A 108.454,B 90.000,C 0.000} C_DIS
LIN {X 91.701,Y -275.120,Z 143.268,A 108.434,B 90.000,C 0.000} C_DIS
LIN {X 91.186,Y -275.291,Z 143.676,A 108.327,B 90.000,C 0.000} C_DIS
LIN {X 90.896,Y -275.387,Z 143.795,A 108.266,B 90.000,C 0.000} C_DIS
LIN {X 90.745,Y -275.437,Z 143.926,A 108.235,B 90.000,C 0.000} C_DIS
LIN {X 90.552,Y -275.500,Z 144.044,A 108.195,B 90.000,C 0.000} C_DIS
LIN {X 89.823,Y -275.739,Z 144.361,A 108.043,B 90.000,C 0.000} C_DIS
LIN {X 89.783,Y -275.752,Z 144.403,A 108.035,B 90.000,C 0.000} C_DIS
LIN {X 89.404,Y -275.875,Z 144.577,A 107.956,B 90.000,C 0.000} C_DIS
LIN {X 89.133,Y -275.962,Z 144.745,A 107.900,B 90.000,C 0.000} C_DIS
LIN {X 88.917,Y -276.032,Z 144.805,A 107.855,B 90.000,C 0.000} C_DIS
LIN {X 87.864,Y -276.369,Z 145.183,A 107.637,B 90.000,C 0.000} C_DIS
LIN {X 85.483,Y -277.111,Z 145.359,A 107.144,B 90.000,C 0.000} C_DIS
LIN {X 83.091,Y -277.838,Z 145.366,A 106.650,B 90.000,C 0.000} C_DIS
LIN {X 80.698,Y -278.546,Z 145.229,A 106.157,B 90.000,C 0.000} C_DIS
LIN {X 78.348,Y -279.216,Z 144.701,A 105.674,B 90.000,C 0.000} C_DIS
LIN {X 76.028,Y -279.857,Z 144.025,A 105.199,B 90.000,C 0.000} C_DIS
LIN {X 73.732,Y -280.470,Z 143.251,A 104.729,B 90.000,C 0.000} C_DIS
LIN {X 71.936,Y -280.936,Z 142.734,A 104.363,B 90.000,C 0.000} C_DIS
LIN {X 71.315,Y -281.095,Z 142.415,A 104.236,B 90.000,C 0.000} C_DIS
LIN {X 69.126,Y -281.641,Z 141.338,A 103.790,B 90.000,C 0.000} C_DIS
LIN {X 69.033,Y -281.664,Z 141.297,A 103.771,B 90.000,C 0.000} C_DIS
LIN {X 68.912,Y -281.693,Z 141.220,A 103.747,B 90.000,C 0.000} C_DIS
LIN {X 68.807,Y -281.719,Z 141.120,A 103.725,B 90.000,C 0.000} C_DIS
LIN {X 68.624,Y -281.764,Z 139.897,A 103.688,B 90.000,C 0.000} C_DIS
LIN {X 68.498,Y -281.794,Z 137.400,A 103.662,B 90.000,C 0.000} C_DIS
LIN {X 68.519,Y -281.789,Z 134.901,A 103.667,B 90.000,C 0.000} C_DIS
